SPLINE
SPL {X  -106.708, Y  +258.294, Z    +0.000, E1   +53.789, E3 +25392.422}
SPL {X  -137.973, Y  +296.505, Z    +0.000, E1   +48.844, E3 +25431.202}
SPL {X  -154.359, Y  +335.426, Z    +0.000, E1   +34.338, E3 +25444.098}
SPL {X  -159.279, Y  +362.429, Z    +0.000, E1   +16.013, E3 +25447.698}
SPL {X  -159.976, Y  +375.387, Z    +0.000, E1    +4.229, E3 +25448.348}
SPL {X  -159.990, Y  +379.485, Z    +0.000, E1    +0.028, E3 +25448.394}
SPL {X  -159.990, Y  +381.270, Z    +0.000, E1    -3.383, E3 +25448.411}
SPL {X  -159.990, Y  +384.811, Z    +0.000, E1   -11.531, E3 +25448.501}
SPL {X  -159.990, Y  +388.002, Z    +0.000, E1   -19.281, E3 +25448.651}
SPL {X  -159.990, Y  +394.075, Z    +0.000, E1   -32.836, E3 +25449.129}
SPL {X  -159.990, Y  +405.152, Z    +0.000, E1   -50.697, E3 +25450.553}
SPL {X  -159.990, Y  +423.293, Z    +0.000, E1   -63.280, E3 +25454.554}
SPL {X  -159.990, Y  +493.649, Z    +0.000, E1   -71.671, E3 +25480.258}
SPL {X  -159.990, Y  +662.531, Z    +0.000, E1   -73.010, E3 +25567.081}
SPL {X  -159.805, Y  +684.185, Z    +0.000, E1   -72.979, E3 +25581.365}
SPL {X  -158.739, Y  +696.464, Z    +0.000, E1   -72.862, E3 +25590.484}
SPL {X  -156.417, Y  +710.124, Z    +0.000, E1   -72.650, E3 +25601.707}
SPL {X  -153.206, Y  +722.596, Z    +0.000, E1   -72.287, E3 +25613.146}
SPL {X  -150.445, Y  +730.933, Z    +0.000, E1   -71.979, E3 +25621.356}
SPL {X  -147.389, Y  +738.737, Z    +0.000, E1   -71.634, E3 +25629.429}
SPL {X  -144.044, Y  +746.129, Z    +0.000, E1   -71.236, E3 +25637.423}
SPL {X  -140.684, Y  +752.689, Z    +0.000, E1   -70.820, E3 +25644.798}
SPL {X  -137.335, Y  +758.572, Z    +0.000, E1   -70.388, E3 +25651.606}
SPL {X  -134.566, Y  +763.037, Z    +0.000, E1   -70.007, E3 +25656.902}
SPL {X  -131.456, Y  +767.693, Z    +0.000, E1   -69.587, E3 +25662.465}
SPL {X  -127.440, Y  +773.226, Z    +0.000, E1   -69.006, E3 +25669.149}
SPL {X  -123.127, Y  +778.659, Z    +0.000, E1   -68.349, E3 +25675.691}
SPL {X   -80.879, Y  +814.541, Z    +0.000, E1   -55.704, E3 +25798.595}
ENDSPLINE

SPLINE
SPL {X  -125.518, Y  +775.707, Z    +0.000, E1   -52.189, E3 +25970.073}
SPL {X  -150.797, Y  +729.951, Z    +0.000, E1   -39.777, E3 +25992.808}
SPL {X  -158.456, Y  +698.602, Z    +0.000, E1   -21.523, E3 +25998.510}
SPL {X  -159.738, Y  +685.469, Z    +0.000, E1   -10.595, E3 +25999.565}
SPL {X  -159.986, Y  +677.650, Z    +0.000, E1    -3.291, E3 +25999.819}
SPL {X  -159.990, Y  +674.500, Z    +0.000, E1    +0.000, E3 +25999.850}
SPL {X  -159.990, Y  +672.716, Z    +0.000, E1    +3.405, E3 +25999.866}
SPL {X  -159.990, Y  +668.521, Z    +0.000, E1   +13.007, E3 +25999.985}
SPL {X  -159.990, Y  +662.839, Z    +0.000, E1   +26.519, E3 +26000.328}
SPL {X  -159.990, Y  +653.836, Z    +0.000, E1   +43.967, E3 +26001.258}
SPL {X  -159.990, Y  +641.022, Z    +0.000, E1   +57.726, E3 +26003.567}
SPL {X  -159.990, Y  +617.987, Z    +0.000, E1   +67.134, E3 +26009.463}
SPL {X  -159.990, Y  +532.407, Z    +0.000, E1   +73.084, E3 +26040.369}
SPL {X  -159.990, Y  +382.957, Z    +0.000, E1   +73.647, E3 +26116.629}
SPL {X  -159.615, Y  +366.548, Z    +0.000, E1   +73.602, E3 +26127.271}
SPL {X  -157.928, Y  +351.899, Z    +0.000, E1   +73.451, E3 +26138.126}
ENDSPLINE

SPLINE
SPL {X  -159.990, Y  +380.170, Z    +0.000, E1   +69.785, E3 +26154.266}
ENDSPLINE

SPLINE
SPL {X  -158.227, Y  +353.814, Z    +0.000, E1   +70.663, E3 +26166.159}
SPL {X  -155.560, Y  +340.111, Z    +0.000, E1   +70.976, E3 +26173.181}
SPL {X  -151.918, Y  +327.322, Z    +0.000, E1   +71.266, E3 +26179.525}
SPL {X  -144.697, Y  +309.238, Z    +0.000, E1   +71.848, E3 +26186.475}
SPL {X  -140.298, Y  +300.601, Z    +0.000, E1   +71.461, E3 +26194.762}
SPL {X  -137.001, Y  +294.872, Z    +0.000, E1   +71.048, E3 +26201.270}
SPL {X  -133.301, Y  +289.026, Z    +0.000, E1   +70.567, E3 +26208.057}
SPL {X  -128.648, Y  +282.387, Z    +0.000, E1   +69.939, E3 +26215.872}
SPL {X  -125.063, Y  +277.720, Z    +0.000, E1   +69.378, E3 +26221.448}
SPL {X  -122.086, Y  +274.099, Z    +0.000, E1   +68.932, E3 +26225.693}
SPL {X   -84.117, Y  +241.407, Z    +0.000, E1   +58.224, E3 +26316.576}
ENDSPLINE

SPLINE
SPL {X  -106.708, Y  +258.294, Z    +0.000, E1   +53.789, E3 +26495.363}
SPL {X  -137.973, Y  +296.505, Z    +0.000, E1   +48.844, E3 +26534.143}
SPL {X  -154.359, Y  +335.426, Z    +0.000, E1   +34.338, E3 +26547.039}
SPL {X  -159.279, Y  +362.429, Z    +0.000, E1   +16.013, E3 +26550.639}
SPL {X  -159.976, Y  +375.387, Z    +0.000, E1    +4.229, E3 +26551.290}
SPL {X  -159.990, Y  +379.485, Z    +0.000, E1    +0.028, E3 +26551.335}
SPL {X  -159.990, Y  +381.270, Z    +0.000, E1    -3.383, E3 +26551.352}
SPL {X  -159.990, Y  +384.811, Z    +0.000, E1   -11.531, E3 +26551.442}
SPL {X  -159.990, Y  +390.180, Z    +0.000, E1   -24.142, E3 +26551.745}
SPL {X  -159.990, Y  +397.074, Z    +0.000, E1   -39.012, E3 +26552.355}
SPL {X  -159.990, Y  +405.152, Z    +0.000, E1   -50.697, E3 +26553.494}
SPL {X  -159.990, Y  +423.293, Z    +0.000, E1   -63.280, E3 +26557.496}
SPL {X  -159.990, Y  +493.649, Z    +0.000, E1   -71.671, E3 +26583.199}
SPL {X  -159.990, Y  +654.929, Z    +0.000, E1   -72.988, E3 +26665.149}
SPL {X  -159.990, Y  +668.018, Z    +0.000, E1   -72.989, E3 +26673.642}
SPL {X  -159.805, Y  +684.185, Z    +0.000, E1   -72.979, E3 +26684.307}
SPL {X  -158.295, Y  +699.729, Z    +0.000, E1   -72.830, E3 +26695.977}
SPL {X  -155.857, Y  +712.630, Z    +0.000, E1   -72.572, E3 +26706.906}
SPL {X  -153.206, Y  +722.596, Z    +0.000, E1   -72.287, E3 +26716.087}
SPL {X  -150.445, Y  +730.933, Z    +0.000, E1   -71.979, E3 +26724.297}
SPL {X  -147.389, Y  +738.737, Z    +0.000, E1   -71.634, E3 +26732.370}
SPL {X  -144.044, Y  +746.129, Z    +0.000, E1   -71.236, E3 +26740.364}
SPL {X  -140.684, Y  +752.689, Z    +0.000, E1   -70.820, E3 +26747.740}
SPL {X  -137.335, Y  +758.572, Z    +0.000, E1   -70.388, E3 +26754.547}
SPL {X  -133.651, Y  +764.444, Z    +0.000, E1   -69.897, E3 +26761.499}
SPL {X  -130.650, Y  +768.844, Z    +0.000, E1   -69.455, E3 +26766.820}
SPL {X  -127.440, Y  +773.226, Z    +0.000, E1   -69.006, E3 +26772.090}
SPL {X  -123.127, Y  +778.659, Z    +0.000, E1   -68.349, E3 +26778.632}
SPL {X   -80.879, Y  +814.541, Z    +0.000, E1   -55.704, E3 +26901.536}
ENDSPLINE

SPLINE
SPL {X  -125.518, Y  +775.707, Z    +0.000, E1   -52.189, E3 +27073.014}
SPL {X  -150.797, Y  +729.951, Z    +0.000, E1   -39.777, E3 +27095.749}
SPL {X  -157.402, Y  +705.160, Z    +0.000, E1   -26.108, E3 +27100.701}
SPL {X  -159.480, Y  +689.270, Z    +0.000, E1   -14.023, E3 +27102.266}
SPL {X  -159.986, Y  +677.650, Z    +0.000, E1    -3.291, E3 +27102.761}
SPL {X  -159.990, Y  +674.500, Z    +0.000, E1    +0.000, E3 +27102.791}
SPL {X  -159.990, Y  +672.716, Z    +0.000, E1    +3.405, E3 +27102.808}
SPL {X  -159.990, Y  +668.521, Z    +0.000, E1   +13.007, E3 +27102.927}
SPL {X  -159.990, Y  +664.286, Z    +0.000, E1   +23.338, E3 +27103.158}
SPL {X  -159.990, Y  +658.431, Z    +0.000, E1   +35.998, E3 +27103.653}
SPL {X  -159.990, Y  +650.524, Z    +0.000, E1   +48.779, E3 +27104.641}
SPL {X  -159.990, Y  +641.022, Z    +0.000, E1   +57.726, E3 +27106.508}
SPL {X  -159.990, Y  +617.987, Z    +0.000, E1   +67.134, E3 +27112.404}
SPL {X  -159.990, Y  +532.407, Z    +0.000, E1   +73.084, E3 +27143.310}
SPL {X  -159.990, Y  +390.607, Z    +0.000, E1   +73.632, E3 +27214.847}
SPL {X  -159.886, Y  +371.742, Z    +0.000, E1   +73.650, E3 +27226.633}
SPL {X  -157.928, Y  +351.899, Z    +0.000, E1   +73.451, E3 +27241.067}
ENDSPLINE

SPLINE
SPL {X  -159.990, Y  +380.170, Z    +0.000, E1   +69.785, E3 +27257.207}
ENDSPLINE

SPLINE
SPL {X  -158.227, Y  +353.814, Z    +0.000, E1   +70.663, E3 +27269.101}
SPL {X  -154.257, Y  +335.055, Z    +0.000, E1   +71.089, E3 +27278.729}
SPL {X  -148.153, Y  +317.104, Z    +0.000, E1   +71.658, E3 +27285.874}
SPL {X  -143.479, Y  +306.716, Z    +0.000, E1   +71.847, E3 +27290.948}
SPL {X  -140.298, Y  +300.601, Z    +0.000, E1   +71.461, E3 +27297.703}
SPL {X  -137.001, Y  +294.872, Z    +0.000, E1   +71.048, E3 +27304.212}
SPL {X  -133.301, Y  +289.026, Z    +0.000, E1   +70.567, E3 +27310.998}
SPL {X  -129.603, Y  +283.692, Z    +0.000, E1   +70.051, E3 +27317.298}
SPL {X  -125.807, Y  +278.659, Z    +0.000, E1   +69.508, E3 +27323.257}
SPL {X  -122.086, Y  +274.099, Z    +0.000, E1   +68.932, E3 +27328.634}
SPL {X   -84.117, Y  +241.407, Z    +0.000, E1   +58.224, E3 +27419.517}
ENDSPLINE

SPLINE
SPL {X  -116.986, Y  +268.362, Z    +0.000, E1   +53.233, E3 +27613.432}
SPL {X  -146.319, Y  +312.789, Z    +0.000, E1   +44.152, E3 +27643.899}
SPL {X  -157.053, Y  +346.986, Z    +0.000, E1   +27.437, E3 +27651.930}
SPL {X  -159.518, Y  +365.226, Z    +0.000, E1   +13.562, E3 +27653.795}
SPL {X  -159.976, Y  +375.387, Z    +0.000, E1    +4.229, E3 +27654.231}
SPL {X  -159.990, Y  +379.485, Z    +0.000, E1    +0.028, E3 +27654.276}
SPL {X  -159.990, Y  +381.270, Z    +0.000, E1    -3.383, E3 +27654.293}
SPL {X  -159.990, Y  +384.811, Z    +0.000, E1   -11.531, E3 +27654.383}
SPL {X  -159.990, Y  +390.180, Z    +0.000, E1   -24.142, E3 +27654.686}
SPL {X  -159.990, Y  +397.074, Z    +0.000, E1   -39.012, E3 +27655.296}
SPL {X  -159.990, Y  +405.152, Z    +0.000, E1   -50.697, E3 +27656.435}
SPL {X  -159.990, Y  +423.293, Z    +0.000, E1   -63.280, E3 +27660.437}
SPL {X  -159.990, Y  +493.649, Z    +0.000, E1   -71.671, E3 +27686.141}
SPL {X  -159.990, Y  +662.531, Z    +0.000, E1   -73.010, E3 +27772.964}
SPL {X  -159.805, Y  +684.185, Z    +0.000, E1   -72.979, E3 +27787.248}
SPL {X  -158.295, Y  +699.729, Z    +0.000, E1   -72.830, E3 +27798.918}
SPL {X  -155.857, Y  +712.630, Z    +0.000, E1   -72.572, E3 +27809.847}
SPL {X  -153.206, Y  +722.596, Z    +0.000, E1   -72.287, E3 +27819.028}
SPL {X  -150.445, Y  +730.933, Z    +0.000, E1   -71.979, E3 +27827.238}
SPL {X  -147.389, Y  +738.737, Z    +0.000, E1   -71.634, E3 +27835.311}
SPL {X  -144.044, Y  +746.129, Z    +0.000, E1   -71.236, E3 +27843.305}
SPL {X  -140.684, Y  +752.689, Z    +0.000, E1   -70.820, E3 +27850.681}
SPL {X  -137.335, Y  +758.572, Z    +0.000, E1   -70.388, E3 +27857.488}
SPL {X  -133.651, Y  +764.444, Z    +0.000, E1   -69.897, E3 +27864.440}
SPL {X  -129.492, Y  +770.461, Z    +0.000, E1   -69.311, E3 +27871.680}
SPL {X  -125.168, Y  +776.148, Z    +0.000, E1   -68.666, E3 +27878.557}
SPL {X  -122.036, Y  +779.960, Z    +0.000, E1   -68.144, E3 +27883.160}
SPL {X   -80.879, Y  +814.541, Z    +0.000, E1   -55.704, E3 +28004.478}
ENDSPLINE

SPLINE
SPL {X  -125.518, Y  +775.707, Z    +0.000, E1   -52.189, E3 +28175.955}
SPL {X  -144.748, Y  +744.653, Z    +0.000, E1   -45.208, E3 +28194.151}
SPL {X  -153.147, Y  +722.791, Z    +0.000, E1   -36.417, E3 +28200.547}
SPL {X  -157.402, Y  +705.160, Z    +0.000, E1   -26.108, E3 +28203.642}
SPL {X  -159.480, Y  +689.270, Z    +0.000, E1   -14.023, E3 +28205.208}
SPL {X  -159.986, Y  +677.650, Z    +0.000, E1    -3.291, E3 +28205.702}
SPL {X  -159.990, Y  +674.500, Z    +0.000, E1    +0.000, E3 +28205.732}
SPL {X  -159.990, Y  +672.716, Z    +0.000, E1    +3.405, E3 +28205.749}
SPL {X  -159.990, Y  +668.521, Z    +0.000, E1   +13.007, E3 +28205.868}
SPL {X  -159.990, Y  +664.286, Z    +0.000, E1   +23.338, E3 +28206.099}
SPL {X  -159.990, Y  +658.431, Z    +0.000, E1   +35.998, E3 +28206.594}
SPL {X  -159.990, Y  +650.524, Z    +0.000, E1   +48.779, E3 +28207.582}
SPL {X  -159.990, Y  +641.022, Z    +0.000, E1   +57.726, E3 +28209.449}
SPL {X  -159.990, Y  +617.987, Z    +0.000, E1   +67.134, E3 +28215.345}
SPL {X  -159.990, Y  +532.407, Z    +0.000, E1   +73.084, E3 +28246.252}
SPL {X  -159.990, Y  +390.607, Z    +0.000, E1   +73.632, E3 +28317.788}
SPL {X  -159.886, Y  +371.742, Z    +0.000, E1   +73.650, E3 +28329.574}
SPL {X  -157.928, Y  +351.899, Z    +0.000, E1   +73.451, E3 +28344.008}
ENDSPLINE

SPLINE
SPL {X  -159.990, Y  +380.170, Z    +0.000, E1   +69.785, E3 +28360.148}
ENDSPLINE

SPLINE
SPL {X  -158.227, Y  +353.814, Z    +0.000, E1   +70.663, E3 +28372.042}
SPL {X  -155.560, Y  +340.111, Z    +0.000, E1   +70.976, E3 +28379.064}
SPL {X  -151.918, Y  +327.322, Z    +0.000, E1   +71.266, E3 +28385.407}
SPL {X  -144.697, Y  +309.238, Z    +0.000, E1   +71.848, E3 +28392.357}
SPL {X  -140.298, Y  +300.601, Z    +0.000, E1   +71.461, E3 +28400.644}
SPL {X  -137.001, Y  +294.872, Z    +0.000, E1   +71.048, E3 +28407.153}
SPL {X  -133.301, Y  +289.026, Z    +0.000, E1   +70.567, E3 +28413.939}
SPL {X  -129.603, Y  +283.692, Z    +0.000, E1   +70.051, E3 +28420.239}
SPL {X  -125.807, Y  +278.659, Z    +0.000, E1   +69.508, E3 +28426.198}
SPL {X  -122.086, Y  +274.099, Z    +0.000, E1   +68.932, E3 +28431.576}
SPL {X   -84.117, Y  +241.407, Z    +0.000, E1   +58.224, E3 +28522.458}
ENDSPLINE

SPLINE
SPL {X  -106.708, Y  +258.294, Z    +0.000, E1   +53.789, E3 +28701.245}
SPL {X  -137.973, Y  +296.505, Z    +0.000, E1   +48.844, E3 +28740.025}
SPL {X  -154.359, Y  +335.426, Z    +0.000, E1   +34.338, E3 +28752.921}
SPL {X  -159.279, Y  +362.429, Z    +0.000, E1   +16.013, E3 +28756.521}
SPL {X  -159.976, Y  +375.387, Z    +0.000, E1    +4.229, E3 +28757.172}
SPL {X  -159.990, Y  +379.485, Z    +0.000, E1    +0.028, E3 +28757.217}
SPL {X  -159.990, Y  +381.270, Z    +0.000, E1    -3.383, E3 +28757.234}
SPL {X  -159.990, Y  +386.246, Z    +0.000, E1   -14.704, E3 +28757.392}
SPL {X  -159.990, Y  +394.075, Z    +0.000, E1   -32.836, E3 +28757.952}
SPL {X  -159.990, Y  +405.152, Z    +0.000, E1   -50.697, E3 +28759.377}
SPL {X  -159.990, Y  +423.293, Z    +0.000, E1   -63.280, E3 +28763.378}
SPL {X  -159.990, Y  +493.649, Z    +0.000, E1   -71.671, E3 +28789.082}
SPL {X  -159.990, Y  +662.531, Z    +0.000, E1   -73.010, E3 +28875.905}
SPL {X  -159.805, Y  +684.185, Z    +0.000, E1   -72.979, E3 +28890.189}
SPL {X  -158.295, Y  +699.729, Z    +0.000, E1   -72.830, E3 +28901.859}
SPL {X  -155.857, Y  +712.630, Z    +0.000, E1   -72.572, E3 +28912.788}
SPL {X  -153.206, Y  +722.596, Z    +0.000, E1   -72.287, E3 +28921.969}
SPL {X  -150.445, Y  +730.933, Z    +0.000, E1   -71.979, E3 +28930.179}
SPL {X  -147.389, Y  +738.737, Z    +0.000, E1   -71.634, E3 +28938.252}
SPL {X  -144.044, Y  +746.129, Z    +0.000, E1   -71.236, E3 +28946.247}
SPL {X  -140.684, Y  +752.689, Z    +0.000, E1   -70.820, E3 +28953.622}
SPL {X  -136.099, Y  +760.606, Z    +0.000, E1   -70.253, E3 +28962.777}
SPL {X  -131.456, Y  +767.693, Z    +0.000, E1   -69.587, E3 +28971.289}
SPL {X  -127.440, Y  +773.226, Z    +0.000, E1   -69.006, E3 +28977.973}
SPL {X  -123.127, Y  +778.659, Z    +0.000, E1   -68.349, E3 +28984.515}
SPL {X   -80.879, Y  +814.541, Z    +0.000, E1   -55.704, E3 +29107.419}
ENDSPLINE

SPLINE
SPL {X  -125.518, Y  +775.707, Z    +0.000, E1   -52.189, E3 +29278.896}
SPL {X  -150.797, Y  +729.951, Z    +0.000, E1   -39.777, E3 +29301.631}
SPL {X  -157.402, Y  +705.160, Z    +0.000, E1   -26.108, E3 +29306.583}
SPL {X  -159.480, Y  +689.270, Z    +0.000, E1   -14.023, E3 +29308.149}
SPL {X  -159.986, Y  +677.650, Z    +0.000, E1    -3.291, E3 +29308.643}
SPL {X  -159.990, Y  +674.500, Z    +0.000, E1    +0.000, E3 +29308.673}
SPL {X  -159.990, Y  +672.716, Z    +0.000, E1    +3.405, E3 +29308.690}
SPL {X  -159.990, Y  +668.521, Z    +0.000, E1   +13.007, E3 +29308.809}
SPL {X  -159.990, Y  +662.839, Z    +0.000, E1   +26.519, E3 +29309.151}
SPL {X  -159.990, Y  +653.836, Z    +0.000, E1   +43.967, E3 +29310.082}
SPL {X  -159.990, Y  +641.022, Z    +0.000, E1   +57.726, E3 +29312.391}
SPL {X  -159.990, Y  +617.987, Z    +0.000, E1   +67.134, E3 +29318.286}
SPL {X  -159.990, Y  +532.407, Z    +0.000, E1   +73.084, E3 +29349.193}
SPL {X  -159.990, Y  +390.607, Z    +0.000, E1   +73.632, E3 +29420.729}
SPL {X  -159.886, Y  +371.742, Z    +0.000, E1   +73.650, E3 +29432.516}
SPL {X  -157.928, Y  +351.899, Z    +0.000, E1   +73.451, E3 +29446.949}
ENDSPLINE

SPLINE
SPL {X  -159.990, Y  +380.170, Z    +0.000, E1   +69.785, E3 +29463.089}
ENDSPLINE

SPLINE
SPL {X  -158.227, Y  +353.814, Z    +0.000, E1   +70.663, E3 +29474.983}
SPL {X  -155.560, Y  +340.111, Z    +0.000, E1   +70.976, E3 +29482.005}
SPL {X  -151.918, Y  +327.322, Z    +0.000, E1   +71.266, E3 +29488.349}
SPL {X  -144.697, Y  +309.238, Z    +0.000, E1   +71.848, E3 +29495.298}
SPL {X  -140.298, Y  +300.601, Z    +0.000, E1   +71.461, E3 +29503.586}
SPL {X  -135.903, Y  +293.078, Z    +0.000, E1   +70.930, E3 +29512.123}
SPL {X  -130.487, Y  +284.926, Z    +0.000, E1   +70.202, E3 +29521.683}
SPL {X  -125.807, Y  +278.659, Z    +0.000, E1   +69.508, E3 +29529.139}
SPL {X  -122.967, Y  +275.148, Z    +0.000, E1   +69.053, E3 +29533.308}
SPL {X  -121.236, Y  +273.103, Z    +0.000, E1   +68.779, E3 +29535.694}
SPL {X   -84.117, Y  +241.407, Z    +0.000, E1   +58.224, E3 +29625.399}
ENDSPLINE

SPLINE
SPL {X  -116.986, Y  +268.362, Z    +0.000, E1   +53.233, E3 +29819.315}
SPL {X  -146.319, Y  +312.789, Z    +0.000, E1   +44.152, E3 +29849.781}
SPL {X  -157.053, Y  +346.986, Z    +0.000, E1   +27.437, E3 +29857.812}
SPL {X  -159.518, Y  +365.226, Z    +0.000, E1   +13.562, E3 +29859.678}
SPL {X  -159.976, Y  +375.387, Z    +0.000, E1    +4.229, E3 +29860.113}
SPL {X  -159.990, Y  +379.485, Z    +0.000, E1    +0.028, E3 +29860.158}
SPL {X  -159.990, Y  +381.270, Z    +0.000, E1    -3.383, E3 +29860.175}
SPL {X  -159.990, Y  +386.246, Z    +0.000, E1   -14.704, E3 +29860.333}
SPL {X  -159.990, Y  +394.075, Z    +0.000, E1   -32.836, E3 +29860.894}
SPL {X  -159.990, Y  +405.152, Z    +0.000, E1   -50.697, E3 +29862.318}
SPL {X  -159.990, Y  +423.293, Z    +0.000, E1   -63.280, E3 +29866.319}
SPL {X  -159.990, Y  +493.649, Z    +0.000, E1   -71.671, E3 +29892.023}
SPL {X  -159.990, Y  +662.531, Z    +0.000, E1   -73.010, E3 +29978.846}
SPL {X  -159.805, Y  +684.185, Z    +0.000, E1   -72.979, E3 +29993.130}
SPL {X  -158.295, Y  +699.729, Z    +0.000, E1   -72.830, E3 +30004.800}
SPL {X  -155.857, Y  +712.630, Z    +0.000, E1   -72.572, E3 +30015.729}
SPL {X  -153.206, Y  +722.596, Z    +0.000, E1   -72.287, E3 +30024.910}
SPL {X  -150.445, Y  +730.933, Z    +0.000, E1   -71.979, E3 +30033.121}
SPL {X  -147.389, Y  +738.737, Z    +0.000, E1   -71.634, E3 +30041.193}
SPL {X  -144.044, Y  +746.129, Z    +0.000, E1   -71.236, E3 +30049.188}
SPL {X  -140.684, Y  +752.689, Z    +0.000, E1   -70.820, E3 +30056.563}
SPL {X  -136.099, Y  +760.606, Z    +0.000, E1   -70.253, E3 +30065.718}
SPL {X  -131.456, Y  +767.693, Z    +0.000, E1   -69.587, E3 +30074.230}
SPL {X  -127.440, Y  +773.226, Z    +0.000, E1   -69.006, E3 +30080.914}
SPL {X  -123.127, Y  +778.659, Z    +0.000, E1   -68.349, E3 +30087.456}
SPL {X   -80.879, Y  +814.541, Z    +0.000, E1   -55.704, E3 +30210.360}
ENDSPLINE

SPLINE
SPL {X  -125.518, Y  +775.707, Z    +0.000, E1   -52.189, E3 +30381.837}
SPL {X  -150.797, Y  +729.951, Z    +0.000, E1   -39.777, E3 +30404.572}
SPL {X  -158.456, Y  +698.602, Z    +0.000, E1   -21.523, E3 +30410.275}
SPL {X  -159.738, Y  +685.469, Z    +0.000, E1   -10.595, E3 +30411.329}
SPL {X  -159.986, Y  +677.650, Z    +0.000, E1    -3.291, E3 +30411.584}
SPL {X  -159.990, Y  +674.500, Z    +0.000, E1    +0.000, E3 +30411.615}
SPL {X  -159.990, Y  +672.716, Z    +0.000, E1    +3.405, E3 +30411.631}
SPL {X  -159.990, Y  +668.521, Z    +0.000, E1   +13.007, E3 +30411.750}
SPL {X  -159.990, Y  +662.839, Z    +0.000, E1   +26.519, E3 +30412.093}
SPL {X  -159.990, Y  +653.836, Z    +0.000, E1   +43.967, E3 +30413.023}
SPL {X  -159.990, Y  +641.022, Z    +0.000, E1   +57.726, E3 +30415.332}
SPL {X  -159.990, Y  +617.987, Z    +0.000, E1   +67.134, E3 +30421.227}
SPL {X  -159.990, Y  +532.407, Z    +0.000, E1   +73.084, E3 +30452.134}
SPL {X  -159.990, Y  +382.957, Z    +0.000, E1   +73.647, E3 +30528.394}
SPL {X  -159.615, Y  +366.548, Z    +0.000, E1   +73.602, E3 +30539.036}
SPL {X  -157.928, Y  +351.899, Z    +0.000, E1   +73.451, E3 +30549.890}
ENDSPLINE

SPLINE
SPL {X  -159.990, Y  +380.170, Z    +0.000, E1   +69.785, E3 +30566.031}
ENDSPLINE

SPLINE
SPL {X  -158.227, Y  +353.814, Z    +0.000, E1   +70.663, E3 +30577.924}
SPL {X  -154.257, Y  +335.055, Z    +0.000, E1   +71.089, E3 +30587.552}
SPL {X  -148.153, Y  +317.104, Z    +0.000, E1   +71.658, E3 +30594.698}
SPL {X  -143.479, Y  +306.716, Z    +0.000, E1   +71.847, E3 +30599.771}
SPL {X  -140.298, Y  +300.601, Z    +0.000, E1   +71.461, E3 +30606.527}
SPL {X  -137.001, Y  +294.872, Z    +0.000, E1   +71.048, E3 +30613.035}
SPL {X  -133.301, Y  +289.026, Z    +0.000, E1   +70.567, E3 +30619.822}
SPL {X  -128.648, Y  +282.387, Z    +0.000, E1   +69.939, E3 +30627.637}
SPL {X  -125.063, Y  +277.720, Z    +0.000, E1   +69.378, E3 +30633.213}
SPL {X  -122.086, Y  +274.099, Z    +0.000, E1   +68.932, E3 +30637.458}
SPL {X   -84.117, Y  +241.407, Z    +0.000, E1   +58.224, E3 +30728.341}
ENDSPLINE

SPLINE
SPL {X  -106.708, Y  +258.294, Z    +0.000, E1   +53.789, E3 +30907.127}
SPL {X  -137.973, Y  +296.505, Z    +0.000, E1   +48.844, E3 +30945.908}
SPL {X  -154.359, Y  +335.426, Z    +0.000, E1   +34.338, E3 +30958.804}
SPL {X  -159.279, Y  +362.429, Z    +0.000, E1   +16.013, E3 +30962.404}
SPL {X  -159.976, Y  +375.387, Z    +0.000, E1    +4.229, E3 +30963.054}
SPL {X  -159.990, Y  +379.485, Z    +0.000, E1    +0.028, E3 +30963.099}
SPL {X  -159.990, Y  +381.270, Z    +0.000, E1    -3.383, E3 +30963.117}
SPL {X  -159.990, Y  +384.811, Z    +0.000, E1   -11.531, E3 +30963.207}
SPL {X  -159.990, Y  +390.180, Z    +0.000, E1   -24.142, E3 +30963.510}
SPL {X  -159.990, Y  +397.074, Z    +0.000, E1   -39.012, E3 +30964.120}
SPL {X  -159.990, Y  +405.152, Z    +0.000, E1   -50.697, E3 +30965.259}
SPL {X  -159.990, Y  +423.293, Z    +0.000, E1   -63.280, E3 +30969.260}
SPL {X  -159.990, Y  +493.649, Z    +0.000, E1   -71.671, E3 +30994.964}
SPL {X  -159.990, Y  +662.531, Z    +0.000, E1   -73.010, E3 +31081.787}
SPL {X  -159.805, Y  +684.185, Z    +0.000, E1   -72.979, E3 +31096.071}
SPL {X  -158.739, Y  +696.464, Z    +0.000, E1   -72.862, E3 +31105.190}
SPL {X  -156.417, Y  +710.124, Z    +0.000, E1   -72.650, E3 +31116.413}
SPL {X  -153.206, Y  +722.596, Z    +0.000, E1   -72.287, E3 +31127.851}
SPL {X  -150.445, Y  +730.933, Z    +0.000, E1   -71.979, E3 +31136.062}
SPL {X  -147.389, Y  +738.737, Z    +0.000, E1   -71.634, E3 +31144.135}
SPL {X  -144.044, Y  +746.129, Z    +0.000, E1   -71.236, E3 +31152.129}
SPL {X  -140.684, Y  +752.689, Z    +0.000, E1   -70.820, E3 +31159.504}
SPL {X  -137.335, Y  +758.572, Z    +0.000, E1   -70.388, E3 +31166.311}
SPL {X  -134.566, Y  +763.037, Z    +0.000, E1   -70.007, E3 +31171.608}
SPL {X  -131.456, Y  +767.693, Z    +0.000, E1   -69.587, E3 +31177.171}
SPL {X  -127.440, Y  +773.226, Z    +0.000, E1   -69.006, E3 +31183.855}
SPL {X  -123.127, Y  +778.659, Z    +0.000, E1   -68.349, E3 +31190.397}
SPL {X   -80.879, Y  +814.541, Z    +0.000, E1   -55.704, E3 +31313.301}
ENDSPLINE

SPLINE
SPL {X  -125.518, Y  +775.707, Z    +0.000, E1   -52.189, E3 +31484.779}
SPL {X  -144.748, Y  +744.653, Z    +0.000, E1   -45.208, E3 +31502.974}
SPL {X  -153.147, Y  +722.791, Z    +0.000, E1   -36.417, E3 +31509.370}
SPL {X  -157.402, Y  +705.160, Z    +0.000, E1   -26.108, E3 +31512.465}
SPL {X  -159.480, Y  +689.270, Z    +0.000, E1   -14.023, E3 +31514.031}
SPL {X  -159.986, Y  +677.650, Z    +0.000, E1    -3.291, E3 +31514.525}
SPL {X  -159.990, Y  +674.500, Z    +0.000, E1    +0.000, E3 +31514.556}
SPL {X  -159.990, Y  +672.716, Z    +0.000, E1    +3.405, E3 +31514.572}
SPL {X  -159.990, Y  +668.521, Z    +0.000, E1   +13.007, E3 +31514.691}
SPL {X  -159.990, Y  +662.839, Z    +0.000, E1   +26.519, E3 +31515.034}
SPL {X  -159.990, Y  +653.836, Z    +0.000, E1   +43.967, E3 +31515.964}
SPL {X  -159.990, Y  +641.022, Z    +0.000, E1   +57.726, E3 +31518.273}
SPL {X  -159.990, Y  +617.987, Z    +0.000, E1   +67.134, E3 +31524.168}
SPL {X  -159.990, Y  +532.407, Z    +0.000, E1   +73.084, E3 +31555.075}
SPL {X  -159.990, Y  +382.957, Z    +0.000, E1   +73.647, E3 +31631.335}
SPL {X  -159.615, Y  +366.548, Z    +0.000, E1   +73.602, E3 +31641.977}
SPL {X  -157.928, Y  +351.899, Z    +0.000, E1   +73.451, E3 +31652.832}
ENDSPLINE

SPLINE
SPL {X  -159.990, Y  +380.170, Z    +0.000, E1   +69.785, E3 +31668.972}
ENDSPLINE

SPLINE
SPL {X  -158.227, Y  +353.814, Z    +0.000, E1   +70.663, E3 +31680.865}
SPL {X  -155.560, Y  +340.111, Z    +0.000, E1   +70.976, E3 +31687.887}
SPL {X  -151.918, Y  +327.322, Z    +0.000, E1   +71.266, E3 +31694.231}
SPL {X  -144.697, Y  +309.238, Z    +0.000, E1   +71.848, E3 +31701.181}
SPL {X  -140.298, Y  +300.601, Z    +0.000, E1   +71.461, E3 +31709.468}
SPL {X  -135.903, Y  +293.078, Z    +0.000, E1   +70.930, E3 +31718.006}
SPL {X  -130.487, Y  +284.926, Z    +0.000, E1   +70.202, E3 +31727.565}
SPL {X  -125.807, Y  +278.659, Z    +0.000, E1   +69.508, E3 +31735.022}
SPL {X  -122.967, Y  +275.148, Z    +0.000, E1   +69.053, E3 +31739.190}
SPL {X  -121.236, Y  +273.103, Z    +0.000, E1   +68.779, E3 +31741.576}
SPL {X   -84.117, Y  +241.407, Z    +0.000, E1   +58.224, E3 +31831.282}
ENDSPLINE

SPLINE
SPL {X  -106.708, Y  +258.294, Z    +0.000, E1   +53.789, E3 +32010.069}
SPL {X  -137.973, Y  +296.505, Z    +0.000, E1   +48.844, E3 +32048.849}
SPL {X  -150.692, Y  +323.752, Z    +0.000, E1   +39.895, E3 +32059.214}
SPL {X  -157.053, Y  +346.986, Z    +0.000, E1   +27.437, E3 +32063.695}
SPL {X  -159.518, Y  +365.226, Z    +0.000, E1   +13.562, E3 +32065.560}
SPL {X  -159.976, Y  +375.387, Z    +0.000, E1    +4.229, E3 +32065.996}
SPL {X  -159.990, Y  +379.485, Z    +0.000, E1    +0.028, E3 +32066.041}
SPL {X  -159.990, Y  +381.270, Z    +0.000, E1    -3.383, E3 +32066.058}
SPL {X  -159.990, Y  +384.811, Z    +0.000, E1   -11.531, E3 +32066.148}
SPL {X  -159.990, Y  +390.180, Z    +0.000, E1   -24.142, E3 +32066.451}
SPL {X  -159.990, Y  +397.074, Z    +0.000, E1   -39.012, E3 +32067.061}
SPL {X  -159.990, Y  +405.152, Z    +0.000, E1   -50.697, E3 +32068.200}
SPL {X  -159.990, Y  +423.293, Z    +0.000, E1   -63.280, E3 +32072.201}
SPL {X  -159.990, Y  +493.649, Z    +0.000, E1   -71.671, E3 +32097.905}
SPL {X  -159.990, Y  +662.531, Z    +0.000, E1   -73.010, E3 +32184.728}
SPL {X  -159.805, Y  +684.185, Z    +0.000, E1   -72.979, E3 +32199.012}
SPL {X  -158.739, Y  +696.464, Z    +0.000, E1   -72.862, E3 +32208.131}
SPL {X  -156.417, Y  +710.124, Z    +0.000, E1   -72.650, E3 +32219.355}
SPL {X  -153.206, Y  +722.596, Z    +0.000, E1   -72.287, E3 +32230.793}
SPL {X  -150.445, Y  +730.933, Z    +0.000, E1   -71.979, E3 +32239.003}
SPL {X  -147.389, Y  +738.737, Z    +0.000, E1   -71.634, E3 +32247.076}
SPL {X  -144.044, Y  +746.129, Z    +0.000, E1   -71.236, E3 +32255.070}
SPL {X  -140.684, Y  +752.689, Z    +0.000, E1   -70.820, E3 +32262.445}
SPL {X  -137.335, Y  +758.572, Z    +0.000, E1   -70.388, E3 +32269.253}
SPL {X  -133.651, Y  +764.444, Z    +0.000, E1   -69.897, E3 +32276.205}
SPL {X  -129.492, Y  +770.461, Z    +0.000, E1   -69.311, E3 +32283.445}
SPL {X  -125.168, Y  +776.148, Z    +0.000, E1   -68.666, E3 +32290.321}
SPL {X  -122.036, Y  +779.960, Z    +0.000, E1   -68.144, E3 +32294.925}
SPL {X   -80.879, Y  +814.541, Z    +0.000, E1   -55.704, E3 +32416.242}
ENDSPLINE

SPLINE
SPL {X  -125.518, Y  +775.707, Z    +0.000, E1   -52.189, E3 +32587.720}
SPL {X  -144.748, Y  +744.653, Z    +0.000, E1   -45.208, E3 +32605.916}
SPL {X  -153.147, Y  +722.791, Z    +0.000, E1   -36.417, E3 +32612.311}
SPL {X  -158.456, Y  +698.602, Z    +0.000, E1   -21.523, E3 +32616.157}
SPL {X  -159.738, Y  +685.469, Z    +0.000, E1   -10.595, E3 +32617.212}
SPL {X  -159.986, Y  +677.650, Z    +0.000, E1    -3.291, E3 +32617.467}
SPL {X  -159.990, Y  +674.500, Z    +0.000, E1    +0.000, E3 +32617.497}
SPL {X  -159.990, Y  +672.716, Z    +0.000, E1    +3.405, E3 +32617.513}
SPL {X  -159.990, Y  +668.521, Z    +0.000, E1   +13.007, E3 +32617.633}
SPL {X  -159.990, Y  +662.839, Z    +0.000, E1   +26.519, E3 +32617.975}
SPL {X  -159.990, Y  +653.836, Z    +0.000, E1   +43.967, E3 +32618.905}
SPL {X  -159.990, Y  +641.022, Z    +0.000, E1   +57.726, E3 +32621.214}
SPL {X  -159.990, Y  +617.987, Z    +0.000, E1   +67.134, E3 +32627.110}
SPL {X  -159.990, Y  +532.407, Z    +0.000, E1   +73.084, E3 +32658.016}
SPL {X  -159.990, Y  +382.957, Z    +0.000, E1   +73.647, E3 +32734.276}
SPL {X  -159.615, Y  +366.548, Z    +0.000, E1   +73.602, E3 +32744.918}
SPL {X  -157.928, Y  +351.899, Z    +0.000, E1   +73.451, E3 +32755.773}
ENDSPLINE

SPLINE
SPL {X  -159.990, Y  +380.170, Z    +0.000, E1   +69.785, E3 +32771.913}
ENDSPLINE

SPLINE
SPL {X  -158.227, Y  +353.814, Z    +0.000, E1   +70.663, E3 +32783.806}
SPL {X  -155.560, Y  +340.111, Z    +0.000, E1   +70.976, E3 +32790.829}
SPL {X  -151.918, Y  +327.322, Z    +0.000, E1   +71.266, E3 +32797.172}
SPL {X  -144.697, Y  +309.238, Z    +0.000, E1   +71.848, E3 +32804.122}
SPL {X  -140.298, Y  +300.601, Z    +0.000, E1   +71.461, E3 +32812.409}
SPL {X  -135.903, Y  +293.078, Z    +0.000, E1   +70.930, E3 +32820.947}
SPL {X  -132.382, Y  +287.656, Z    +0.000, E1   +70.425, E3 +32827.339}
SPL {X  -128.648, Y  +282.387, Z    +0.000, E1   +69.939, E3 +32833.519}
SPL {X  -125.063, Y  +277.720, Z    +0.000, E1   +69.378, E3 +32839.095}
SPL {X  -122.086, Y  +274.099, Z    +0.000, E1   +68.932, E3 +32843.340}
SPL {X   -84.117, Y  +241.407, Z    +0.000, E1   +58.224, E3 +32934.223}
ENDSPLINE

SPLINE
SPL {X  -116.986, Y  +268.362, Z    +0.000, E1   +53.233, E3 +33128.138}
SPL {X  -146.319, Y  +312.789, Z    +0.000, E1   +44.152, E3 +33158.604}
SPL {X  -155.980, Y  +341.904, Z    +0.000, E1   +30.583, E3 +33165.900}
SPL {X  -159.279, Y  +362.429, Z    +0.000, E1   +16.013, E3 +33168.286}
SPL {X  -159.976, Y  +375.387, Z    +0.000, E1    +4.229, E3 +33168.937}
SPL {X  -159.990, Y  +379.485, Z    +0.000, E1    +0.028, E3 +33168.982}
SPL {X  -159.990, Y  +381.270, Z    +0.000, E1    -3.383, E3 +33168.999}
SPL {X  -159.990, Y  +386.246, Z    +0.000, E1   -14.704, E3 +33169.156}
SPL {X  -159.990, Y  +394.075, Z    +0.000, E1   -32.836, E3 +33169.717}
SPL {X  -159.990, Y  +405.152, Z    +0.000, E1   -50.697, E3 +33171.141}
SPL {X  -159.990, Y  +423.293, Z    +0.000, E1   -63.280, E3 +33175.143}
SPL {X  -159.990, Y  +493.649, Z    +0.000, E1   -71.671, E3 +33200.847}
SPL {X  -159.990, Y  +662.531, Z    +0.000, E1   -73.010, E3 +33287.670}
SPL {X  -159.805, Y  +684.185, Z    +0.000, E1   -72.979, E3 +33301.954}
SPL {X  -158.295, Y  +699.729, Z    +0.000, E1   -72.830, E3 +33313.624}
SPL {X  -155.857, Y  +712.630, Z    +0.000, E1   -72.572, E3 +33324.553}
SPL {X  -153.206, Y  +722.596, Z    +0.000, E1   -72.287, E3 +33333.734}
SPL {X  -150.445, Y  +730.933, Z    +0.000, E1   -71.979, E3 +33341.944}
SPL {X  -147.389, Y  +738.737, Z    +0.000, E1   -71.634, E3 +33350.017}
SPL {X  -144.044, Y  +746.129, Z    +0.000, E1   -71.236, E3 +33358.011}
SPL {X  -140.684, Y  +752.689, Z    +0.000, E1   -70.820, E3 +33365.387}
SPL {X  -137.335, Y  +758.572, Z    +0.000, E1   -70.388, E3 +33372.194}
SPL {X  -133.651, Y  +764.444, Z    +0.000, E1   -69.897, E3 +33379.146}
SPL {X  -129.492, Y  +770.461, Z    +0.000, E1   -69.311, E3 +33386.386}
SPL {X  -125.168, Y  +776.148, Z    +0.000, E1   -68.666, E3 +33393.262}
SPL {X  -122.036, Y  +779.960, Z    +0.000, E1   -68.144, E3 +33397.866}
SPL {X   -80.879, Y  +814.541, Z    +0.000, E1   -55.704, E3 +33519.184}
ENDSPLINE

SPLINE
SPL {X  -125.518, Y  +775.707, Z    +0.000, E1   -52.189, E3 +33690.661}
SPL {X  -144.748, Y  +744.653, Z    +0.000, E1   -45.208, E3 +33708.857}
SPL {X  -153.147, Y  +722.791, Z    +0.000, E1   -36.417, E3 +33715.252}
SPL {X  -157.402, Y  +705.160, Z    +0.000, E1   -26.108, E3 +33718.348}
SPL {X  -159.480, Y  +689.270, Z    +0.000, E1   -14.023, E3 +33719.913}
SPL {X  -159.986, Y  +677.650, Z    +0.000, E1    -3.291, E3 +33720.408}
SPL {X  -159.990, Y  +674.500, Z    +0.000, E1    +0.000, E3 +33720.438}
SPL {X  -159.990, Y  +672.716, Z    +0.000, E1    +3.405, E3 +33720.455}
SPL {X  -159.990, Y  +668.521, Z    +0.000, E1   +13.007, E3 +33720.574}
SPL {X  -159.990, Y  +664.286, Z    +0.000, E1   +23.338, E3 +33720.805}
SPL {X  -159.990, Y  +658.431, Z    +0.000, E1   +35.998, E3 +33721.300}
SPL {X  -159.990, Y  +650.524, Z    +0.000, E1   +48.779, E3 +33722.288}
SPL {X  -159.990, Y  +641.022, Z    +0.000, E1   +57.726, E3 +33724.155}
SPL {X  -159.990, Y  +617.987, Z    +0.000, E1   +67.134, E3 +33730.051}
SPL {X  -159.990, Y  +532.407, Z    +0.000, E1   +73.084, E3 +33760.957}
SPL {X  -159.990, Y  +390.607, Z    +0.000, E1   +73.632, E3 +33832.494}
SPL {X  -159.886, Y  +371.742, Z    +0.000, E1   +73.650, E3 +33844.280}
SPL {X  -157.928, Y  +351.899, Z    +0.000, E1   +73.451, E3 +33858.714}
ENDSPLINE

SPLINE
SPL {X  -159.990, Y  +380.170, Z    +0.000, E1   +69.785, E3 +33874.854}
ENDSPLINE

SPLINE
SPL {X  -158.227, Y  +353.814, Z    +0.000, E1   +70.663, E3 +33886.748}
SPL {X  -155.560, Y  +340.111, Z    +0.000, E1   +70.976, E3 +33893.770}
SPL {X  -151.918, Y  +327.322, Z    +0.000, E1   +71.266, E3 +33900.113}
SPL {X  -144.697, Y  +309.238, Z    +0.000, E1   +71.848, E3 +33907.063}
SPL {X  -140.298, Y  +300.601, Z    +0.000, E1   +71.461, E3 +33915.350}
SPL {X  -137.001, Y  +294.872, Z    +0.000, E1   +71.048, E3 +33921.859}
SPL {X  -133.301, Y  +289.026, Z    +0.000, E1   +70.567, E3 +33928.645}
SPL {X  -129.603, Y  +283.692, Z    +0.000, E1   +70.051, E3 +33934.945}
SPL {X  -125.807, Y  +278.659, Z    +0.000, E1   +69.508, E3 +33940.904}
SPL {X  -122.086, Y  +274.099, Z    +0.000, E1   +68.932, E3 +33946.281}
SPL {X   -84.117, Y  +241.407, Z    +0.000, E1   +58.224, E3 +34037.164}
ENDSPLINE

SPLINE
SPL {X  -116.986, Y  +268.362, Z    +0.000, E1   +53.233, E3 +34231.080}
SPL {X  -146.319, Y  +312.789, Z    +0.000, E1   +44.152, E3 +34261.546}
SPL {X  -157.053, Y  +346.986, Z    +0.000, E1   +27.437, E3 +34269.577}
SPL {X  -159.518, Y  +365.226, Z    +0.000, E1   +13.562, E3 +34271.442}
SPL {X  -159.976, Y  +375.387, Z    +0.000, E1    +4.229, E3 +34271.878}
SPL {X  -159.990, Y  +379.485, Z    +0.000, E1    +0.028, E3 +34271.923}
SPL {X  -159.990, Y  +381.270, Z    +0.000, E1    -3.383, E3 +34271.940}
SPL {X  -159.990, Y  +386.246, Z    +0.000, E1   -14.704, E3 +34272.098}
SPL {X  -159.990, Y  +394.075, Z    +0.000, E1   -32.836, E3 +34272.658}
SPL {X  -159.990, Y  +405.152, Z    +0.000, E1   -50.697, E3 +34274.082}
SPL {X  -159.990, Y  +423.293, Z    +0.000, E1   -63.280, E3 +34278.084}
SPL {X  -159.990, Y  +493.649, Z    +0.000, E1   -71.671, E3 +34303.788}
SPL {X  -159.990, Y  +662.531, Z    +0.000, E1   -73.010, E3 +34390.611}
SPL {X  -159.805, Y  +684.185, Z    +0.000, E1   -72.979, E3 +34404.895}
SPL {X  -158.295, Y  +699.729, Z    +0.000, E1   -72.830, E3 +34416.565}
SPL {X  -155.857, Y  +712.630, Z    +0.000, E1   -72.572, E3 +34427.494}
SPL {X  -153.206, Y  +722.596, Z    +0.000, E1   -72.287, E3 +34436.675}
SPL {X  -150.445, Y  +730.933, Z    +0.000, E1   -71.979, E3 +34444.885}
SPL {X  -147.389, Y  +738.737, Z    +0.000, E1   -71.634, E3 +34452.958}
SPL {X  -144.044, Y  +746.129, Z    +0.000, E1   -71.236, E3 +34460.952}
SPL {X  -140.684, Y  +752.689, Z    +0.000, E1   -70.820, E3 +34468.328}
SPL {X  -136.099, Y  +760.606, Z    +0.000, E1   -70.253, E3 +34477.483}
SPL {X  -131.456, Y  +767.693, Z    +0.000, E1   -69.587, E3 +34485.995}
SPL {X  -128.507, Y  +771.803, Z    +0.000, E1   -69.145, E3 +34490.977}
SPL {X  -125.168, Y  +776.148, Z    +0.000, E1   -68.666, E3 +34496.204}
SPL {X  -122.036, Y  +779.960, Z    +0.000, E1   -68.144, E3 +34500.807}
SPL {X   -80.879, Y  +814.541, Z    +0.000, E1   -55.704, E3 +34622.125}
ENDSPLINE

SPLINE
SPL {X  -125.518, Y  +775.707, Z    +0.000, E1   -52.189, E3 +34793.602}
SPL {X  -150.797, Y  +729.951, Z    +0.000, E1   -39.777, E3 +34816.337}
SPL {X  -158.456, Y  +698.602, Z    +0.000, E1   -21.523, E3 +34822.040}
SPL {X  -159.738, Y  +685.469, Z    +0.000, E1   -10.595, E3 +34823.094}
SPL {X  -159.986, Y  +677.650, Z    +0.000, E1    -3.291, E3 +34823.349}
SPL {X  -159.990, Y  +674.500, Z    +0.000, E1    +0.000, E3 +34823.379}
SPL {X  -159.990, Y  +672.716, Z    +0.000, E1    +3.405, E3 +34823.396}
SPL {X  -159.990, Y  +668.521, Z    +0.000, E1   +13.007, E3 +34823.515}
SPL {X  -159.990, Y  +662.839, Z    +0.000, E1   +26.519, E3 +34823.857}
SPL {X  -159.990, Y  +653.836, Z    +0.000, E1   +43.967, E3 +34824.787}
SPL {X  -159.990, Y  +641.022, Z    +0.000, E1   +57.726, E3 +34827.096}
SPL {X  -159.990, Y  +617.987, Z    +0.000, E1   +67.134, E3 +34832.992}
SPL {X  -159.990, Y  +532.407, Z    +0.000, E1   +73.084, E3 +34863.899}
SPL {X  -159.990, Y  +382.957, Z    +0.000, E1   +73.647, E3 +34940.158}
SPL {X  -159.615, Y  +366.548, Z    +0.000, E1   +73.602, E3 +34950.801}
SPL {X  -157.928, Y  +351.899, Z    +0.000, E1   +73.451, E3 +34961.655}
ENDSPLINE

SPLINE
SPL {X  -159.990, Y  +380.170, Z    +0.000, E1   +69.785, E3 +34977.795}
ENDSPLINE

SPLINE
SPL {X  -158.227, Y  +353.814, Z    +0.000, E1   +70.663, E3 +34989.689}
SPL {X  -155.560, Y  +340.111, Z    +0.000, E1   +70.976, E3 +34996.711}
SPL {X  -151.918, Y  +327.322, Z    +0.000, E1   +71.266, E3 +35003.054}
SPL {X  -144.697, Y  +309.238, Z    +0.000, E1   +71.848, E3 +35010.004}
SPL {X  -140.298, Y  +300.601, Z    +0.000, E1   +71.461, E3 +35018.292}
SPL {X  -137.001, Y  +294.872, Z    +0.000, E1   +71.048, E3 +35024.800}
SPL {X  -133.301, Y  +289.026, Z    +0.000, E1   +70.567, E3 +35031.586}
SPL {X  -128.648, Y  +282.387, Z    +0.000, E1   +69.939, E3 +35039.402}
SPL {X  -125.063, Y  +277.720, Z    +0.000, E1   +69.378, E3 +35044.977}
SPL {X  -122.086, Y  +274.099, Z    +0.000, E1   +68.932, E3 +35049.223}
SPL {X   -84.117, Y  +241.407, Z    +0.000, E1   +58.224, E3 +35140.105}
ENDSPLINE

SPLINE
SPL {X  -106.708, Y  +258.294, Z    +0.000, E1   +53.789, E3 +35318.892}
SPL {X  -137.973, Y  +296.505, Z    +0.000, E1   +48.844, E3 +35357.672}
SPL {X  -154.359, Y  +335.426, Z    +0.000, E1   +34.338, E3 +35370.568}
SPL {X  -159.279, Y  +362.429, Z    +0.000, E1   +16.013, E3 +35374.168}
SPL {X  -159.976, Y  +375.387, Z    +0.000, E1    +4.229, E3 +35374.819}
SPL {X  -159.990, Y  +379.485, Z    +0.000, E1    +0.028, E3 +35374.864}
SPL {X  -159.990, Y  +381.270, Z    +0.000, E1    -3.383, E3 +35374.881}
SPL {X  -159.990, Y  +384.811, Z    +0.000, E1   -11.531, E3 +35374.971}
SPL {X  -159.990, Y  +390.180, Z    +0.000, E1   -24.142, E3 +35375.274}
SPL {X  -159.990, Y  +397.074, Z    +0.000, E1   -39.012, E3 +35375.884}
SPL {X  -159.990, Y  +405.152, Z    +0.000, E1   -50.697, E3 +35377.024}
SPL {X  -159.990, Y  +423.293, Z    +0.000, E1   -63.280, E3 +35381.025}
SPL {X  -159.990, Y  +493.649, Z    +0.000, E1   -71.671, E3 +35406.729}
SPL {X  -159.990, Y  +654.929, Z    +0.000, E1   -72.988, E3 +35488.679}
SPL {X  -159.990, Y  +668.018, Z    +0.000, E1   -72.989, E3 +35497.171}
SPL {X  -159.805, Y  +684.185, Z    +0.000, E1   -72.979, E3 +35507.836}
SPL {X  -158.295, Y  +699.729, Z    +0.000, E1   -72.830, E3 +35519.506}
SPL {X  -155.857, Y  +712.630, Z    +0.000, E1   -72.572, E3 +35530.435}
SPL {X  -153.206, Y  +722.596, Z    +0.000, E1   -72.287, E3 +35539.616}
SPL {X  -150.445, Y  +730.933, Z    +0.000, E1   -71.979, E3 +35547.827}
SPL {X  -147.389, Y  +738.737, Z    +0.000, E1   -71.634, E3 +35555.899}
SPL {X  -144.044, Y  +746.129, Z    +0.000, E1   -71.236, E3 +35563.894}
SPL {X  -140.684, Y  +752.689, Z    +0.000, E1   -70.820, E3 +35571.269}
SPL {X  -136.099, Y  +760.606, Z    +0.000, E1   -70.253, E3 +35580.424}
SPL {X  -131.456, Y  +767.693, Z    +0.000, E1   -69.587, E3 +35588.936}
SPL {X  -128.507, Y  +771.803, Z    +0.000, E1   -69.145, E3 +35593.918}
SPL {X  -125.168, Y  +776.148, Z    +0.000, E1   -68.666, E3 +35599.145}
SPL {X  -122.036, Y  +779.960, Z    +0.000, E1   -68.144, E3 +35603.748}
SPL {X   -80.879, Y  +814.541, Z    +0.000, E1   -55.704, E3 +35725.066}
ENDSPLINE

SPLINE
SPL {X  -125.518, Y  +775.707, Z    +0.000, E1   -52.189, E3 +35896.543}
SPL {X  -150.797, Y  +729.951, Z    +0.000, E1   -39.777, E3 +35919.278}
SPL {X  -157.402, Y  +705.160, Z    +0.000, E1   -26.108, E3 +35924.230}
SPL {X  -159.480, Y  +689.270, Z    +0.000, E1   -14.023, E3 +35925.796}
SPL {X  -159.986, Y  +677.650, Z    +0.000, E1    -3.291, E3 +35926.290}
SPL {X  -159.990, Y  +674.500, Z    +0.000, E1    +0.000, E3 +35926.320}
SPL {X  -159.990, Y  +672.716, Z    +0.000, E1    +3.405, E3 +35926.337}
SPL {X  -159.990, Y  +668.521, Z    +0.000, E1   +13.007, E3 +35926.456}
SPL {X  -159.990, Y  +662.839, Z    +0.000, E1   +26.519, E3 +35926.798}
SPL {X  -159.990, Y  +653.836, Z    +0.000, E1   +43.967, E3 +35927.729}
SPL {X  -159.990, Y  +641.022, Z    +0.000, E1   +57.726, E3 +35930.038}
SPL {X  -159.990, Y  +617.987, Z    +0.000, E1   +67.134, E3 +35935.933}
SPL {X  -159.990, Y  +532.407, Z    +0.000, E1   +73.084, E3 +35966.840}
SPL {X  -159.990, Y  +382.957, Z    +0.000, E1   +73.647, E3 +36043.099}
SPL {X  -159.196, Y  +361.585, Z    +0.000, E1   +73.581, E3 +36057.222}
SPL {X  -157.239, Y  +347.958, Z    +0.000, E1   +73.365, E3 +36067.817}
ENDSPLINE

SPLINE
SPL {X  -159.990, Y  +380.170, Z    +0.000, E1   +69.785, E3 +36080.736}
ENDSPLINE

SPLINE
SPL {X  -158.227, Y  +353.814, Z    +0.000, E1   +70.663, E3 +36092.630}
SPL {X  -155.560, Y  +340.111, Z    +0.000, E1   +70.976, E3 +36099.652}
SPL {X  -151.918, Y  +327.322, Z    +0.000, E1   +71.266, E3 +36105.996}
SPL {X  -144.697, Y  +309.238, Z    +0.000, E1   +71.848, E3 +36112.945}
SPL {X  -140.298, Y  +300.601, Z    +0.000, E1   +71.461, E3 +36121.233}
SPL {X  -137.001, Y  +294.872, Z    +0.000, E1   +71.048, E3 +36127.741}
SPL {X  -133.301, Y  +289.026, Z    +0.000, E1   +70.567, E3 +36134.527}
SPL {X  -129.603, Y  +283.692, Z    +0.000, E1   +70.051, E3 +36140.827}
SPL {X  -125.807, Y  +278.659, Z    +0.000, E1   +69.508, E3 +36146.786}
SPL {X  -122.086, Y  +274.099, Z    +0.000, E1   +68.932, E3 +36152.164}
SPL {X   -84.117, Y  +241.407, Z    +0.000, E1   +58.224, E3 +36243.046}
ENDSPLINE

SPLINE
SPL {X  -106.708, Y  +258.294, Z    +0.000, E1   +53.789, E3 +36421.833}
SPL {X  -137.973, Y  +296.505, Z    +0.000, E1   +48.844, E3 +36460.613}
SPL {X  -154.359, Y  +335.426, Z    +0.000, E1   +34.338, E3 +36473.509}
SPL {X  -159.279, Y  +362.429, Z    +0.000, E1   +16.013, E3 +36477.110}
SPL {X  -159.976, Y  +375.387, Z    +0.000, E1    +4.229, E3 +36477.760}
SPL {X  -159.990, Y  +379.485, Z    +0.000, E1    +0.028, E3 +36477.805}
SPL {X  -159.990, Y  +381.270, Z    +0.000, E1    -3.383, E3 +36477.822}
SPL {X  -159.990, Y  +386.246, Z    +0.000, E1   -14.704, E3 +36477.980}
SPL {X  -159.990, Y  +394.075, Z    +0.000, E1   -32.836, E3 +36478.541}
SPL {X  -159.990, Y  +405.152, Z    +0.000, E1   -50.697, E3 +36479.965}
SPL {X  -159.990, Y  +423.293, Z    +0.000, E1   -63.280, E3 +36483.966}
SPL {X  -159.990, Y  +493.649, Z    +0.000, E1   -71.671, E3 +36509.670}
SPL {X  -159.990, Y  +662.531, Z    +0.000, E1   -73.010, E3 +36596.493}
SPL {X  -159.805, Y  +684.185, Z    +0.000, E1   -72.979, E3 +36610.777}
SPL {X  -158.295, Y  +699.729, Z    +0.000, E1   -72.830, E3 +36622.447}
SPL {X  -155.857, Y  +712.630, Z    +0.000, E1   -72.572, E3 +36633.376}
SPL {X  -153.206, Y  +722.596, Z    +0.000, E1   -72.287, E3 +36642.557}
SPL {X  -150.445, Y  +730.933, Z    +0.000, E1   -71.979, E3 +36650.768}
SPL {X  -147.389, Y  +738.737, Z    +0.000, E1   -71.634, E3 +36658.840}
SPL {X  -144.044, Y  +746.129, Z    +0.000, E1   -71.236, E3 +36666.835}
SPL {X  -140.684, Y  +752.689, Z    +0.000, E1   -70.820, E3 +36674.210}
SPL {X  -136.099, Y  +760.606, Z    +0.000, E1   -70.253, E3 +36683.366}
SPL {X  -131.456, Y  +767.693, Z    +0.000, E1   -69.587, E3 +36691.877}
SPL {X  -127.440, Y  +773.226, Z    +0.000, E1   -69.006, E3 +36698.561}
SPL {X  -123.127, Y  +778.659, Z    +0.000, E1   -68.349, E3 +36705.103}
SPL {X   -80.879, Y  +814.541, Z    +0.000, E1   -55.704, E3 +36828.007}
ENDSPLINE

SPLINE
SPL {X  -125.518, Y  +775.707, Z    +0.000, E1   -52.189, E3 +36999.484}
SPL {X  -144.748, Y  +744.653, Z    +0.000, E1   -45.208, E3 +37017.680}
SPL {X  -153.147, Y  +722.791, Z    +0.000, E1   -36.417, E3 +37024.076}
SPL {X  -157.402, Y  +705.160, Z    +0.000, E1   -26.108, E3 +37027.171}
SPL {X  -159.480, Y  +689.270, Z    +0.000, E1   -14.023, E3 +37028.737}
SPL {X  -159.986, Y  +677.650, Z    +0.000, E1    -3.291, E3 +37029.231}
SPL {X  -159.990, Y  +674.500, Z    +0.000, E1    +0.000, E3 +37029.262}
SPL {X  -159.990, Y  +672.716, Z    +0.000, E1    +3.405, E3 +37029.278}
SPL {X  -159.990, Y  +668.521, Z    +0.000, E1   +13.007, E3 +37029.397}
SPL {X  -159.990, Y  +664.286, Z    +0.000, E1   +23.338, E3 +37029.629}
SPL {X  -159.990, Y  +658.431, Z    +0.000, E1   +35.998, E3 +37030.123}
SPL {X  -159.990, Y  +650.524, Z    +0.000, E1   +48.779, E3 +37031.112}
SPL {X  -159.990, Y  +641.022, Z    +0.000, E1   +57.726, E3 +37032.979}
SPL {X  -159.990, Y  +617.987, Z    +0.000, E1   +67.134, E3 +37038.874}
SPL {X  -159.990, Y  +532.407, Z    +0.000, E1   +73.084, E3 +37069.781}
SPL {X  -159.990, Y  +390.607, Z    +0.000, E1   +73.632, E3 +37141.317}
SPL {X  -159.886, Y  +371.742, Z    +0.000, E1   +73.650, E3 +37153.104}
SPL {X  -157.928, Y  +351.899, Z    +0.000, E1   +73.451, E3 +37167.537}
ENDSPLINE

SPLINE
SPL {X  -159.990, Y  +380.170, Z    +0.000, E1   +69.785, E3 +37183.678}
ENDSPLINE

SPLINE
SPL {X  -158.227, Y  +353.814, Z    +0.000, E1   +70.663, E3 +37195.571}
SPL {X  -155.560, Y  +340.111, Z    +0.000, E1   +70.976, E3 +37202.593}
SPL {X  -151.918, Y  +327.322, Z    +0.000, E1   +71.266, E3 +37208.937}
SPL {X  -144.697, Y  +309.238, Z    +0.000, E1   +71.848, E3 +37215.886}
SPL {X  -140.298, Y  +300.601, Z    +0.000, E1   +71.461, E3 +37224.174}
SPL {X  -135.903, Y  +293.078, Z    +0.000, E1   +70.930, E3 +37232.712}
SPL {X  -132.382, Y  +287.656, Z    +0.000, E1   +70.425, E3 +37239.103}
SPL {X  -128.648, Y  +282.387, Z    +0.000, E1   +69.939, E3 +37245.284}
SPL {X  -125.063, Y  +277.720, Z    +0.000, E1   +69.378, E3 +37250.860}
SPL {X  -122.086, Y  +274.099, Z    +0.000, E1   +68.932, E3 +37255.105}
SPL {X   -84.117, Y  +241.407, Z    +0.000, E1   +58.224, E3 +37345.988}
ENDSPLINE

SPLINE
SPL {X  -106.708, Y  +258.294, Z    +0.000, E1   +53.789, E3 +37524.775}
SPL {X  -137.973, Y  +296.505, Z    +0.000, E1   +48.844, E3 +37563.555}
SPL {X  -154.359, Y  +335.426, Z    +0.000, E1   +34.338, E3 +37576.451}
SPL {X  -159.279, Y  +362.429, Z    +0.000, E1   +16.013, E3 +37580.051}
SPL {X  -159.976, Y  +375.387, Z    +0.000, E1    +4.229, E3 +37580.701}
SPL {X  -159.990, Y  +379.485, Z    +0.000, E1    +0.028, E3 +37580.746}
SPL {X  -159.990, Y  +381.270, Z    +0.000, E1    -3.383, E3 +37580.764}
SPL {X  -159.990, Y  +384.811, Z    +0.000, E1   -11.531, E3 +37580.854}
SPL {X  -159.990, Y  +390.180, Z    +0.000, E1   -24.142, E3 +37581.157}
SPL {X  -159.990, Y  +397.074, Z    +0.000, E1   -39.012, E3 +37581.767}
SPL {X  -159.990, Y  +405.152, Z    +0.000, E1   -50.697, E3 +37582.906}
SPL {X  -159.990, Y  +423.293, Z    +0.000, E1   -63.280, E3 +37586.907}
SPL {X  -159.990, Y  +493.649, Z    +0.000, E1   -71.671, E3 +37612.611}
SPL {X  -159.990, Y  +662.531, Z    +0.000, E1   -73.010, E3 +37699.434}
SPL {X  -159.805, Y  +684.185, Z    +0.000, E1   -72.979, E3 +37713.718}
SPL {X  -158.739, Y  +696.464, Z    +0.000, E1   -72.862, E3 +37722.837}
SPL {X  -156.417, Y  +710.124, Z    +0.000, E1   -72.650, E3 +37734.060}
SPL {X  -153.206, Y  +722.596, Z    +0.000, E1   -72.287, E3 +37745.499}
SPL {X  -150.445, Y  +730.933, Z    +0.000, E1   -71.979, E3 +37753.709}
SPL {X  -147.389, Y  +738.737, Z    +0.000, E1   -71.634, E3 +37761.782}
SPL {X  -144.044, Y  +746.129, Z    +0.000, E1   -71.236, E3 +37769.776}
SPL {X  -140.684, Y  +752.689, Z    +0.000, E1   -70.820, E3 +37777.151}
SPL {X  -137.335, Y  +758.572, Z    +0.000, E1   -70.388, E3 +37783.959}
SPL {X  -134.566, Y  +763.037, Z    +0.000, E1   -70.007, E3 +37789.255}
SPL {X  -131.456, Y  +767.693, Z    +0.000, E1   -69.587, E3 +37794.818}
SPL {X  -127.440, Y  +773.226, Z    +0.000, E1   -69.006, E3 +37801.502}
SPL {X  -123.127, Y  +778.659, Z    +0.000, E1   -68.349, E3 +37808.044}
SPL {X   -80.879, Y  +814.541, Z    +0.000, E1   -55.704, E3 +37930.948}
ENDSPLINE

SPLINE
SPL {X  -125.518, Y  +775.707, Z    +0.000, E1   -52.189, E3 +38102.426}
SPL {X  -144.748, Y  +744.653, Z    +0.000, E1   -45.208, E3 +38120.621}
SPL {X  -153.147, Y  +722.791, Z    +0.000, E1   -36.417, E3 +38127.017}
SPL {X  -157.402, Y  +705.160, Z    +0.000, E1   -26.108, E3 +38130.112}
SPL {X  -159.480, Y  +689.270, Z    +0.000, E1   -14.023, E3 +38131.678}
SPL {X  -159.986, Y  +677.650, Z    +0.000, E1    -3.291, E3 +38132.172}
SPL {X  -159.990, Y  +674.500, Z    +0.000, E1    +0.000, E3 +38132.203}
SPL {X  -159.990, Y  +672.716, Z    +0.000, E1    +3.405, E3 +38132.219}
SPL {X  -159.990, Y  +668.521, Z    +0.000, E1   +13.007, E3 +38132.338}
SPL {X  -159.990, Y  +662.839, Z    +0.000, E1   +26.519, E3 +38132.681}
SPL {X  -159.990, Y  +653.836, Z    +0.000, E1   +43.967, E3 +38133.611}
SPL {X  -159.990, Y  +641.022, Z    +0.000, E1   +57.726, E3 +38135.920}
SPL {X  -159.990, Y  +617.987, Z    +0.000, E1   +67.134, E3 +38141.815}
SPL {X  -159.990, Y  +532.407, Z    +0.000, E1   +73.084, E3 +38172.722}
SPL {X  -159.990, Y  +382.957, Z    +0.000, E1   +73.647, E3 +38248.982}
SPL {X  -159.615, Y  +366.548, Z    +0.000, E1   +73.602, E3 +38259.624}
SPL {X  -157.928, Y  +351.899, Z    +0.000, E1   +73.451, E3 +38270.479}
ENDSPLINE

SPLINE
SPL {X  -159.990, Y  +380.170, Z    +0.000, E1   +69.785, E3 +38286.619}
ENDSPLINE

SPLINE
SPL {X  -158.227, Y  +353.814, Z    +0.000, E1   +70.663, E3 +38298.512}
SPL {X  -155.560, Y  +340.111, Z    +0.000, E1   +70.976, E3 +38305.534}
SPL {X  -151.918, Y  +327.322, Z    +0.000, E1   +71.266, E3 +38311.878}
SPL {X  -144.697, Y  +309.238, Z    +0.000, E1   +71.848, E3 +38318.828}
SPL {X  -140.298, Y  +300.601, Z    +0.000, E1   +71.461, E3 +38327.115}
SPL {X  -135.903, Y  +293.078, Z    +0.000, E1   +70.930, E3 +38335.653}
SPL {X  -130.487, Y  +284.926, Z    +0.000, E1   +70.202, E3 +38345.212}
SPL {X  -125.807, Y  +278.659, Z    +0.000, E1   +69.508, E3 +38352.669}
SPL {X  -122.967, Y  +275.148, Z    +0.000, E1   +69.053, E3 +38356.837}
SPL {X  -121.236, Y  +273.103, Z    +0.000, E1   +68.779, E3 +38359.223}
SPL {X   -84.117, Y  +241.407, Z    +0.000, E1   +58.224, E3 +38448.929}
ENDSPLINE

SPLINE
SPL {X  -106.708, Y  +258.294, Z    +0.000, E1   +53.789, E3 +38627.716}
SPL {X  -137.973, Y  +296.505, Z    +0.000, E1   +48.844, E3 +38666.496}
SPL {X  -150.692, Y  +323.752, Z    +0.000, E1   +39.895, E3 +38676.862}
SPL {X  -157.053, Y  +346.986, Z    +0.000, E1   +27.437, E3 +38681.342}
SPL {X  -159.518, Y  +365.226, Z    +0.000, E1   +13.562, E3 +38683.207}
SPL {X  -159.976, Y  +375.387, Z    +0.000, E1    +4.229, E3 +38683.643}
SPL {X  -159.990, Y  +379.485, Z    +0.000, E1    +0.028, E3 +38683.688}
SPL {X  -159.990, Y  +381.270, Z    +0.000, E1    -3.383, E3 +38683.705}
SPL {X  -159.990, Y  +384.811, Z    +0.000, E1   -11.531, E3 +38683.795}
SPL {X  -159.990, Y  +390.180, Z    +0.000, E1   -24.142, E3 +38684.098}
SPL {X  -159.990, Y  +397.074, Z    +0.000, E1   -39.012, E3 +38684.708}
SPL {X  -159.990, Y  +405.152, Z    +0.000, E1   -50.697, E3 +38685.847}
SPL {X  -159.990, Y  +423.293, Z    +0.000, E1   -63.280, E3 +38689.849}
SPL {X  -159.990, Y  +493.649, Z    +0.000, E1   -71.671, E3 +38715.552}
SPL {X  -159.990, Y  +662.531, Z    +0.000, E1   -73.010, E3 +38802.376}
SPL {X  -159.805, Y  +684.185, Z    +0.000, E1   -72.979, E3 +38816.660}
SPL {X  -158.295, Y  +699.729, Z    +0.000, E1   -72.830, E3 +38828.330}
SPL {X  -155.857, Y  +712.630, Z    +0.000, E1   -72.572, E3 +38839.259}
SPL {X  -153.206, Y  +722.596, Z    +0.000, E1   -72.287, E3 +38848.440}
SPL {X  -150.445, Y  +730.933, Z    +0.000, E1   -71.979, E3 +38856.650}
SPL {X  -147.389, Y  +738.737, Z    +0.000, E1   -71.634, E3 +38864.723}
SPL {X  -144.044, Y  +746.129, Z    +0.000, E1   -71.236, E3 +38872.717}
SPL {X  -140.684, Y  +752.689, Z    +0.000, E1   -70.820, E3 +38880.092}
SPL {X  -136.099, Y  +760.606, Z    +0.000, E1   -70.253, E3 +38889.248}
SPL {X  -131.456, Y  +767.693, Z    +0.000, E1   -69.587, E3 +38897.760}
SPL {X  -127.440, Y  +773.226, Z    +0.000, E1   -69.006, E3 +38904.443}
SPL {X  -123.127, Y  +778.659, Z    +0.000, E1   -68.349, E3 +38910.985}
SPL {X   -80.879, Y  +814.541, Z    +0.000, E1   -55.704, E3 +39033.889}
ENDSPLINE

SPLINE
SPL {X  -125.518, Y  +775.707, Z    +0.000, E1   -52.189, E3 +39205.367}
SPL {X  -150.797, Y  +729.951, Z    +0.000, E1   -39.777, E3 +39228.102}
SPL {X  -157.402, Y  +705.160, Z    +0.000, E1   -26.108, E3 +39233.054}
SPL {X  -159.480, Y  +689.270, Z    +0.000, E1   -14.023, E3 +39234.619}
SPL {X  -159.986, Y  +677.650, Z    +0.000, E1    -3.291, E3 +39235.114}
SPL {X  -159.990, Y  +674.500, Z    +0.000, E1    +0.000, E3 +39235.144}
SPL {X  -159.990, Y  +672.716, Z    +0.000, E1    +3.405, E3 +39235.161}
SPL {X  -159.990, Y  +668.521, Z    +0.000, E1   +13.007, E3 +39235.280}
SPL {X  -159.990, Y  +662.839, Z    +0.000, E1   +26.519, E3 +39235.622}
SPL {X  -159.990, Y  +653.836, Z    +0.000, E1   +43.967, E3 +39236.552}
SPL {X  -159.990, Y  +641.022, Z    +0.000, E1   +57.726, E3 +39238.861}
SPL {X  -159.990, Y  +617.987, Z    +0.000, E1   +67.134, E3 +39244.757}
SPL {X  -159.990, Y  +532.407, Z    +0.000, E1   +73.084, E3 +39275.663}
SPL {X  -159.990, Y  +390.607, Z    +0.000, E1   +73.632, E3 +39347.199}
SPL {X  -159.886, Y  +371.742, Z    +0.000, E1   +73.650, E3 +39358.986}
SPL {X  -157.928, Y  +351.899, Z    +0.000, E1   +73.451, E3 +39373.420}
ENDSPLINE

SPLINE
SPL {X  -159.990, Y  +380.170, Z    +0.000, E1   +69.785, E3 +39389.560}
ENDSPLINE

SPLINE
SPL {X  -158.227, Y  +353.814, Z    +0.000, E1   +70.663, E3 +39401.454}
SPL {X  -155.560, Y  +340.111, Z    +0.000, E1   +70.976, E3 +39408.476}
SPL {X  -151.918, Y  +327.322, Z    +0.000, E1   +71.266, E3 +39414.819}
SPL {X  -144.697, Y  +309.238, Z    +0.000, E1   +71.848, E3 +39421.769}
SPL {X  -140.298, Y  +300.601, Z    +0.000, E1   +71.461, E3 +39430.056}
SPL {X  -135.903, Y  +293.078, Z    +0.000, E1   +70.930, E3 +39438.594}
SPL {X  -130.487, Y  +284.926, Z    +0.000, E1   +70.202, E3 +39448.153}
SPL {X  -125.807, Y  +278.659, Z    +0.000, E1   +69.508, E3 +39455.610}
SPL {X  -122.967, Y  +275.148, Z    +0.000, E1   +69.053, E3 +39459.779}
SPL {X  -121.236, Y  +273.103, Z    +0.000, E1   +68.779, E3 +39462.164}
SPL {X   -84.117, Y  +241.407, Z    +0.000, E1   +58.224, E3 +39551.870}
ENDSPLINE

SPLINE
SPL {X  -116.986, Y  +268.362, Z    +0.000, E1   +53.233, E3 +39745.785}
SPL {X  -146.319, Y  +312.789, Z    +0.000, E1   +44.152, E3 +39776.252}
SPL {X  -157.053, Y  +346.986, Z    +0.000, E1   +27.437, E3 +39784.283}
SPL {X  -159.518, Y  +365.226, Z    +0.000, E1   +13.562, E3 +39786.148}
SPL {X  -159.976, Y  +375.387, Z    +0.000, E1    +4.229, E3 +39786.584}
SPL {X  -159.990, Y  +379.485, Z    +0.000, E1    +0.028, E3 +39786.629}
SPL {X  -159.990, Y  +381.270, Z    +0.000, E1    -3.383, E3 +39786.646}
SPL {X  -159.990, Y  +386.246, Z    +0.000, E1   -14.704, E3 +39786.803}
SPL {X  -159.990, Y  +394.075, Z    +0.000, E1   -32.836, E3 +39787.364}
SPL {X  -159.990, Y  +405.152, Z    +0.000, E1   -50.697, E3 +39788.788}
SPL {X  -159.990, Y  +423.293, Z    +0.000, E1   -63.280, E3 +39792.790}
SPL {X  -159.990, Y  +493.649, Z    +0.000, E1   -71.671, E3 +39818.494}
SPL {X  -159.990, Y  +662.531, Z    +0.000, E1   -73.010, E3 +39905.317}
SPL {X  -159.805, Y  +684.185, Z    +0.000, E1   -72.979, E3 +39919.601}
SPL {X  -158.295, Y  +699.729, Z    +0.000, E1   -72.830, E3 +39931.271}
SPL {X  -155.857, Y  +712.630, Z    +0.000, E1   -72.572, E3 +39942.200}
SPL {X  -153.206, Y  +722.596, Z    +0.000, E1   -72.287, E3 +39951.381}
SPL {X  -150.445, Y  +730.933, Z    +0.000, E1   -71.979, E3 +39959.591}
SPL {X  -147.389, Y  +738.737, Z    +0.000, E1   -71.634, E3 +39967.664}
SPL {X  -144.044, Y  +746.129, Z    +0.000, E1   -71.236, E3 +39975.658}
SPL {X  -140.684, Y  +752.689, Z    +0.000, E1   -70.820, E3 +39983.034}
SPL {X  -136.099, Y  +760.606, Z    +0.000, E1   -70.253, E3 +39992.189}
SPL {X  -131.456, Y  +767.693, Z    +0.000, E1   -69.587, E3 +40000.701}
SPL {X  -127.440, Y  +773.226, Z    +0.000, E1   -69.006, E3 +40007.385}
SPL {X  -123.127, Y  +778.659, Z    +0.000, E1   -68.349, E3 +40013.927}
SPL {X   -80.879, Y  +814.541, Z    +0.000, E1   -55.704, E3 +40136.831}
ENDSPLINE

SPLINE
SPL {X  -125.518, Y  +775.707, Z    +0.000, E1   -52.189, E3 +40308.308}
SPL {X  -150.797, Y  +729.951, Z    +0.000, E1   -39.777, E3 +40331.043}
SPL {X  -158.456, Y  +698.602, Z    +0.000, E1   -21.523, E3 +40336.746}
SPL {X  -159.738, Y  +685.469, Z    +0.000, E1   -10.595, E3 +40337.800}
SPL {X  -159.986, Y  +677.650, Z    +0.000, E1    -3.291, E3 +40338.055}
SPL {X  -159.990, Y  +674.500, Z    +0.000, E1    +0.000, E3 +40338.085}
SPL {X  -159.990, Y  +672.716, Z    +0.000, E1    +3.405, E3 +40338.102}
SPL {X  -159.990, Y  +668.521, Z    +0.000, E1   +13.007, E3 +40338.221}
SPL {X  -159.990, Y  +662.839, Z    +0.000, E1   +26.519, E3 +40338.563}
SPL {X  -159.990, Y  +653.836, Z    +0.000, E1   +43.967, E3 +40339.493}
SPL {X  -159.990, Y  +641.022, Z    +0.000, E1   +57.726, E3 +40341.802}
SPL {X  -159.990, Y  +617.987, Z    +0.000, E1   +67.134, E3 +40347.698}
SPL {X  -159.990, Y  +532.407, Z    +0.000, E1   +73.084, E3 +40378.605}
SPL {X  -159.990, Y  +382.957, Z    +0.000, E1   +73.647, E3 +40454.864}
SPL {X  -159.615, Y  +366.548, Z    +0.000, E1   +73.602, E3 +40465.507}
SPL {X  -157.928, Y  +351.899, Z    +0.000, E1   +73.451, E3 +40476.361}
ENDSPLINE

SPLINE
SPL {X  -159.990, Y  +380.170, Z    +0.000, E1   +69.785, E3 +40492.501}
ENDSPLINE

SPLINE
SPL {X  -158.227, Y  +353.814, Z    +0.000, E1   +70.663, E3 +40504.395}
SPL {X  -154.257, Y  +335.055, Z    +0.000, E1   +71.089, E3 +40514.023}
SPL {X  -148.153, Y  +317.104, Z    +0.000, E1   +71.658, E3 +40521.168}
SPL {X  -143.479, Y  +306.716, Z    +0.000, E1   +71.847, E3 +40526.242}
SPL {X  -140.298, Y  +300.601, Z    +0.000, E1   +71.461, E3 +40532.997}
SPL {X  -137.001, Y  +294.872, Z    +0.000, E1   +71.048, E3 +40539.506}
SPL {X  -133.301, Y  +289.026, Z    +0.000, E1   +70.567, E3 +40546.292}
SPL {X  -129.603, Y  +283.692, Z    +0.000, E1   +70.051, E3 +40552.592}
SPL {X  -125.807, Y  +278.659, Z    +0.000, E1   +69.508, E3 +40558.551}
SPL {X  -122.086, Y  +274.099, Z    +0.000, E1   +68.932, E3 +40563.928}
SPL {X   -84.117, Y  +241.407, Z    +0.000, E1   +58.224, E3 +40654.811}
ENDSPLINE

SPLINE
SPL {X  -116.986, Y  +268.362, Z    +0.000, E1   +53.233, E3 +40848.727}
SPL {X  -146.319, Y  +312.789, Z    +0.000, E1   +44.152, E3 +40879.193}
SPL {X  -157.053, Y  +346.986, Z    +0.000, E1   +27.437, E3 +40887.224}
SPL {X  -159.518, Y  +365.226, Z    +0.000, E1   +13.562, E3 +40889.089}
SPL {X  -159.976, Y  +375.387, Z    +0.000, E1    +4.229, E3 +40889.525}
SPL {X  -159.990, Y  +379.485, Z    +0.000, E1    +0.028, E3 +40889.570}
SPL {X  -159.990, Y  +381.270, Z    +0.000, E1    -3.383, E3 +40889.587}
SPL {X  -159.990, Y  +386.246, Z    +0.000, E1   -14.704, E3 +40889.745}
SPL {X  -159.990, Y  +394.075, Z    +0.000, E1   -32.836, E3 +40890.305}
SPL {X  -159.990, Y  +405.152, Z    +0.000, E1   -50.697, E3 +40891.730}
SPL {X  -159.990, Y  +423.293, Z    +0.000, E1   -63.280, E3 +40895.731}
SPL {X  -159.990, Y  +493.649, Z    +0.000, E1   -71.671, E3 +40921.435}
SPL {X  -159.990, Y  +662.531, Z    +0.000, E1   -73.010, E3 +41008.258}
SPL {X  -159.805, Y  +684.185, Z    +0.000, E1   -72.979, E3 +41022.542}
SPL {X  -158.295, Y  +699.729, Z    +0.000, E1   -72.830, E3 +41034.212}
SPL {X  -155.857, Y  +712.630, Z    +0.000, E1   -72.572, E3 +41045.141}
SPL {X  -153.206, Y  +722.596, Z    +0.000, E1   -72.287, E3 +41054.322}
SPL {X  -150.445, Y  +730.933, Z    +0.000, E1   -71.979, E3 +41062.532}
SPL {X  -147.389, Y  +738.737, Z    +0.000, E1   -71.634, E3 +41070.605}
SPL {X  -144.044, Y  +746.129, Z    +0.000, E1   -71.236, E3 +41078.600}
SPL {X  -140.684, Y  +752.689, Z    +0.000, E1   -70.820, E3 +41085.975}
SPL {X  -137.335, Y  +758.572, Z    +0.000, E1   -70.388, E3 +41092.782}
SPL {X  -133.651, Y  +764.444, Z    +0.000, E1   -69.897, E3 +41099.734}
SPL {X  -129.492, Y  +770.461, Z    +0.000, E1   -69.311, E3 +41106.974}
SPL {X  -125.168, Y  +776.148, Z    +0.000, E1   -68.666, E3 +41113.851}
SPL {X  -122.036, Y  +779.960, Z    +0.000, E1   -68.144, E3 +41118.454}
SPL {X   -80.879, Y  +814.541, Z    +0.000, E1   -55.704, E3 +41239.772}
ENDSPLINE

SPLINE
SPL {X  -125.518, Y  +775.707, Z    +0.000, E1   -52.189, E3 +41411.249}
SPL {X  -144.748, Y  +744.653, Z    +0.000, E1   -45.208, E3 +41429.445}
SPL {X  -153.147, Y  +722.791, Z    +0.000, E1   -36.417, E3 +41435.841}
SPL {X  -157.402, Y  +705.160, Z    +0.000, E1   -26.108, E3 +41438.936}
SPL {X  -159.480, Y  +689.270, Z    +0.000, E1   -14.023, E3 +41440.502}
SPL {X  -159.986, Y  +677.650, Z    +0.000, E1    -3.291, E3 +41440.996}
SPL {X  -159.990, Y  +674.500, Z    +0.000, E1    +0.000, E3 +41441.026}
SPL {X  -159.990, Y  +672.716, Z    +0.000, E1    +3.405, E3 +41441.043}
SPL {X  -159.990, Y  +668.521, Z    +0.000, E1   +13.007, E3 +41441.162}
SPL {X  -159.990, Y  +664.286, Z    +0.000, E1   +23.338, E3 +41441.393}
SPL {X  -159.990, Y  +658.431, Z    +0.000, E1   +35.998, E3 +41441.888}
SPL {X  -159.990, Y  +650.524, Z    +0.000, E1   +48.779, E3 +41442.877}
SPL {X  -159.990, Y  +641.022, Z    +0.000, E1   +57.726, E3 +41444.743}
SPL {X  -159.990, Y  +617.987, Z    +0.000, E1   +67.134, E3 +41450.639}
SPL {X  -159.990, Y  +532.407, Z    +0.000, E1   +73.084, E3 +41481.546}
SPL {X  -159.990, Y  +390.607, Z    +0.000, E1   +73.632, E3 +41553.082}
SPL {X  -159.886, Y  +371.742, Z    +0.000, E1   +73.650, E3 +41564.869}
SPL {X  -157.928, Y  +351.899, Z    +0.000, E1   +73.451, E3 +41579.302}
ENDSPLINE

SPLINE
SPL {X  -159.990, Y  +380.170, Z    +0.000, E1   +69.785, E3 +41595.442}
ENDSPLINE

SPLINE
SPL {X  -158.227, Y  +353.814, Z    +0.000, E1   +70.663, E3 +41607.336}
SPL {X  -155.560, Y  +340.111, Z    +0.000, E1   +70.976, E3 +41614.358}
SPL {X  -151.918, Y  +327.322, Z    +0.000, E1   +71.266, E3 +41620.702}
SPL {X  -144.697, Y  +309.238, Z    +0.000, E1   +71.848, E3 +41627.651}
SPL {X  -140.298, Y  +300.601, Z    +0.000, E1   +71.461, E3 +41635.939}
SPL {X  -135.903, Y  +293.078, Z    +0.000, E1   +70.930, E3 +41644.476}
SPL {X  -132.382, Y  +287.656, Z    +0.000, E1   +70.425, E3 +41650.868}
SPL {X  -128.648, Y  +282.387, Z    +0.000, E1   +69.939, E3 +41657.049}
SPL {X  -125.063, Y  +277.720, Z    +0.000, E1   +69.378, E3 +41662.624}
SPL {X  -122.086, Y  +274.099, Z    +0.000, E1   +68.932, E3 +41666.870}
SPL {X   -84.117, Y  +241.407, Z    +0.000, E1   +58.224, E3 +41757.752}
ENDSPLINE

SPLINE
SPL {X  -106.708, Y  +258.294, Z    +0.000, E1   +53.789, E3 +41936.539}
SPL {X  -137.973, Y  +296.505, Z    +0.000, E1   +48.844, E3 +41975.319}
SPL {X  -154.359, Y  +335.426, Z    +0.000, E1   +34.338, E3 +41988.215}
SPL {X  -159.279, Y  +362.429, Z    +0.000, E1   +16.013, E3 +41991.815}
SPL {X  -159.976, Y  +375.387, Z    +0.000, E1    +4.229, E3 +41992.466}
SPL {X  -159.990, Y  +379.485, Z    +0.000, E1    +0.028, E3 +41992.511}
SPL {X  -159.990, Y  +381.270, Z    +0.000, E1    -3.383, E3 +41992.528}
SPL {X  -159.990, Y  +386.246, Z    +0.000, E1   -14.704, E3 +41992.686}
SPL {X  -159.990, Y  +394.075, Z    +0.000, E1   -32.836, E3 +41993.246}
SPL {X  -159.990, Y  +405.152, Z    +0.000, E1   -50.697, E3 +41994.671}
SPL {X  -159.990, Y  +423.293, Z    +0.000, E1   -63.280, E3 +41998.672}
SPL {X  -159.990, Y  +493.649, Z    +0.000, E1   -71.671, E3 +42024.376}
SPL {X  -159.990, Y  +662.531, Z    +0.000, E1   -73.010, E3 +42111.199}
SPL {X  -159.805, Y  +684.185, Z    +0.000, E1   -72.979, E3 +42125.483}
SPL {X  -158.739, Y  +696.464, Z    +0.000, E1   -72.862, E3 +42134.602}
SPL {X  -156.417, Y  +710.124, Z    +0.000, E1   -72.650, E3 +42145.825}
SPL {X  -153.206, Y  +722.596, Z    +0.000, E1   -72.287, E3 +42157.263}
SPL {X  -150.445, Y  +730.933, Z    +0.000, E1   -71.979, E3 +42165.474}
SPL {X  -147.389, Y  +738.737, Z    +0.000, E1   -71.634, E3 +42173.546}
SPL {X  -144.044, Y  +746.129, Z    +0.000, E1   -71.236, E3 +42181.541}
SPL {X  -140.684, Y  +752.689, Z    +0.000, E1   -70.820, E3 +42188.916}
SPL {X  -136.099, Y  +760.606, Z    +0.000, E1   -70.253, E3 +42198.071}
SPL {X  -131.456, Y  +767.693, Z    +0.000, E1   -69.587, E3 +42206.583}
SPL {X  -127.440, Y  +773.226, Z    +0.000, E1   -69.006, E3 +42213.267}
SPL {X  -123.127, Y  +778.659, Z    +0.000, E1   -68.349, E3 +42219.809}
SPL {X   -80.879, Y  +814.541, Z    +0.000, E1   -55.704, E3 +42342.713}
ENDSPLINE

SPLINE
SPL {X  -125.518, Y  +775.707, Z    +0.000, E1   -52.189, E3 +42514.190}
SPL {X  -144.748, Y  +744.653, Z    +0.000, E1   -45.208, E3 +42532.386}
SPL {X  -153.147, Y  +722.791, Z    +0.000, E1   -36.417, E3 +42538.782}
SPL {X  -158.456, Y  +698.602, Z    +0.000, E1   -21.523, E3 +42542.628}
SPL {X  -159.738, Y  +685.469, Z    +0.000, E1   -10.595, E3 +42543.682}
SPL {X  -159.986, Y  +677.650, Z    +0.000, E1    -3.291, E3 +42543.937}
SPL {X  -159.990, Y  +674.500, Z    +0.000, E1    +0.000, E3 +42543.968}
SPL {X  -159.990, Y  +672.716, Z    +0.000, E1    +3.405, E3 +42543.984}
SPL {X  -159.990, Y  +668.521, Z    +0.000, E1   +13.007, E3 +42544.103}
SPL {X  -159.990, Y  +662.839, Z    +0.000, E1   +26.519, E3 +42544.445}
SPL {X  -159.990, Y  +653.836, Z    +0.000, E1   +43.967, E3 +42545.376}
SPL {X  -159.990, Y  +641.022, Z    +0.000, E1   +57.726, E3 +42547.685}
SPL {X  -159.990, Y  +617.987, Z    +0.000, E1   +67.134, E3 +42553.580}
SPL {X  -159.990, Y  +532.407, Z    +0.000, E1   +73.084, E3 +42584.487}
SPL {X  -159.990, Y  +390.607, Z    +0.000, E1   +73.632, E3 +42656.023}
SPL {X  -159.886, Y  +371.742, Z    +0.000, E1   +73.650, E3 +42667.810}
SPL {X  -157.928, Y  +351.899, Z    +0.000, E1   +73.451, E3 +42682.243}
ENDSPLINE

SPLINE
SPL {X  -159.990, Y  +387.996, Z    +0.000, E1   +69.509, E3 +42694.673}
ENDSPLINE

SPLINE
SPL {X  -159.889, Y  +371.819, Z    +0.000, E1   +70.046, E3 +42702.400}
SPL {X  -158.227, Y  +353.814, Z    +0.000, E1   +70.663, E3 +42710.277}
SPL {X  -154.257, Y  +335.055, Z    +0.000, E1   +71.089, E3 +42719.905}
SPL {X  -148.153, Y  +317.104, Z    +0.000, E1   +71.658, E3 +42727.051}
SPL {X  -143.479, Y  +306.716, Z    +0.000, E1   +71.847, E3 +42732.124}
SPL {X  -140.298, Y  +300.601, Z    +0.000, E1   +71.461, E3 +42738.880}
SPL {X  -135.903, Y  +293.078, Z    +0.000, E1   +70.930, E3 +42747.417}
SPL {X  -130.487, Y  +284.926, Z    +0.000, E1   +70.202, E3 +42756.977}
SPL {X  -125.807, Y  +278.659, Z    +0.000, E1   +69.508, E3 +42764.433}
SPL {X  -122.967, Y  +275.148, Z    +0.000, E1   +69.053, E3 +42768.602}
SPL {X  -121.236, Y  +273.103, Z    +0.000, E1   +68.779, E3 +42770.988}
SPL {X   -84.117, Y  +241.407, Z    +0.000, E1   +58.224, E3 +42860.693}
ENDSPLINE

SPLINE
SPL {X  -116.986, Y  +268.362, Z    +0.000, E1   +53.233, E3 +43054.609}
SPL {X  -146.319, Y  +312.789, Z    +0.000, E1   +44.152, E3 +43085.075}
SPL {X  -157.053, Y  +346.986, Z    +0.000, E1   +27.437, E3 +43093.106}
SPL {X  -159.518, Y  +365.226, Z    +0.000, E1   +13.562, E3 +43094.972}
SPL {X  -159.976, Y  +375.387, Z    +0.000, E1    +4.229, E3 +43095.407}
SPL {X  -159.990, Y  +379.485, Z    +0.000, E1    +0.028, E3 +43095.452}
SPL {X  -159.990, Y  +381.270, Z    +0.000, E1    -3.383, E3 +43095.469}
SPL {X  -159.990, Y  +384.811, Z    +0.000, E1   -11.531, E3 +43095.560}
SPL {X  -159.990, Y  +388.002, Z    +0.000, E1   -19.281, E3 +43095.709}
SPL {X  -159.990, Y  +394.075, Z    +0.000, E1   -32.836, E3 +43096.188}
SPL {X  -159.990, Y  +405.152, Z    +0.000, E1   -50.697, E3 +43097.612}
SPL {X  -159.990, Y  +423.293, Z    +0.000, E1   -63.280, E3 +43101.613}
SPL {X  -159.990, Y  +493.649, Z    +0.000, E1   -71.671, E3 +43127.317}
SPL {X  -159.990, Y  +654.929, Z    +0.000, E1   -72.988, E3 +43209.267}
SPL {X  -159.990, Y  +668.018, Z    +0.000, E1   -72.989, E3 +43217.760}
SPL {X  -159.805, Y  +684.185, Z    +0.000, E1   -72.979, E3 +43228.424}
SPL {X  -158.295, Y  +699.729, Z    +0.000, E1   -72.830, E3 +43240.095}
SPL {X  -155.857, Y  +712.630, Z    +0.000, E1   -72.572, E3 +43251.024}
SPL {X  -153.206, Y  +722.596, Z    +0.000, E1   -72.287, E3 +43260.204}
SPL {X  -150.445, Y  +730.933, Z    +0.000, E1   -71.979, E3 +43268.415}
SPL {X  -147.389, Y  +738.737, Z    +0.000, E1   -71.634, E3 +43276.487}
SPL {X  -144.044, Y  +746.129, Z    +0.000, E1   -71.236, E3 +43284.482}
SPL {X  -140.684, Y  +752.689, Z    +0.000, E1   -70.820, E3 +43291.857}
SPL {X  -136.099, Y  +760.606, Z    +0.000, E1   -70.253, E3 +43301.013}
SPL {X  -131.456, Y  +767.693, Z    +0.000, E1   -69.587, E3 +43309.524}
SPL {X  -128.507, Y  +771.803, Z    +0.000, E1   -69.145, E3 +43314.506}
SPL {X  -125.168, Y  +776.148, Z    +0.000, E1   -68.666, E3 +43319.733}
SPL {X  -122.036, Y  +779.960, Z    +0.000, E1   -68.144, E3 +43324.336}
SPL {X   -80.879, Y  +814.541, Z    +0.000, E1   -55.704, E3 +43445.654}
ENDSPLINE

SPLINE
SPL {X  -125.518, Y  +775.707, Z    +0.000, E1   -52.189, E3 +43617.132}
SPL {X  -144.748, Y  +744.653, Z    +0.000, E1   -45.208, E3 +43635.327}
SPL {X  -153.147, Y  +722.791, Z    +0.000, E1   -36.417, E3 +43641.723}
SPL {X  -158.456, Y  +698.602, Z    +0.000, E1   -21.523, E3 +43645.569}
SPL {X  -159.738, Y  +685.469, Z    +0.000, E1   -10.595, E3 +43646.623}
SPL {X  -159.986, Y  +677.650, Z    +0.000, E1    -3.291, E3 +43646.878}
SPL {X  -159.990, Y  +674.500, Z    +0.000, E1    +0.000, E3 +43646.909}
SPL {X  -159.990, Y  +672.716, Z    +0.000, E1    +3.405, E3 +43646.925}
SPL {X  -159.990, Y  +668.521, Z    +0.000, E1   +13.007, E3 +43647.044}
SPL {X  -159.990, Y  +664.286, Z    +0.000, E1   +23.338, E3 +43647.276}
SPL {X  -159.990, Y  +658.431, Z    +0.000, E1   +35.998, E3 +43647.770}
SPL {X  -159.990, Y  +650.524, Z    +0.000, E1   +48.779, E3 +43648.759}
SPL {X  -159.990, Y  +641.022, Z    +0.000, E1   +57.726, E3 +43650.626}
SPL {X  -159.990, Y  +617.987, Z    +0.000, E1   +67.134, E3 +43656.521}
SPL {X  -159.990, Y  +532.407, Z    +0.000, E1   +73.084, E3 +43687.428}
SPL {X  -159.990, Y  +382.957, Z    +0.000, E1   +73.647, E3 +43763.688}
SPL {X  -159.615, Y  +366.548, Z    +0.000, E1   +73.602, E3 +43774.330}
SPL {X  -157.928, Y  +351.899, Z    +0.000, E1   +73.451, E3 +43785.184}
ENDSPLINE

SPLINE
SPL {X  -159.990, Y  +380.170, Z    +0.000, E1   +69.785, E3 +43801.325}
ENDSPLINE

SPLINE
SPL {X  -158.227, Y  +353.814, Z    +0.000, E1   +70.663, E3 +43813.218}
SPL {X  -155.560, Y  +340.111, Z    +0.000, E1   +70.976, E3 +43820.240}
SPL {X  -151.918, Y  +327.322, Z    +0.000, E1   +71.266, E3 +43826.584}
SPL {X  -144.697, Y  +309.238, Z    +0.000, E1   +71.848, E3 +43833.533}
SPL {X  -140.298, Y  +300.601, Z    +0.000, E1   +71.461, E3 +43841.821}
SPL {X  -137.001, Y  +294.872, Z    +0.000, E1   +71.048, E3 +43848.329}
SPL {X  -133.301, Y  +289.026, Z    +0.000, E1   +70.567, E3 +43855.116}
SPL {X  -128.648, Y  +282.387, Z    +0.000, E1   +69.939, E3 +43862.931}
SPL {X  -125.063, Y  +277.720, Z    +0.000, E1   +69.378, E3 +43868.507}
SPL {X  -122.086, Y  +274.099, Z    +0.000, E1   +68.932, E3 +43872.752}
SPL {X   -84.117, Y  +241.407, Z    +0.000, E1   +58.224, E3 +43963.635}
ENDSPLINE

SPLINE
SPL {X  -106.708, Y  +258.294, Z    +0.000, E1   +53.789, E3 +44142.422}
SPL {X  -137.973, Y  +296.505, Z    +0.000, E1   +48.844, E3 +44181.202}
SPL {X  -154.359, Y  +335.426, Z    +0.000, E1   +34.338, E3 +44194.098}
SPL {X  -159.279, Y  +362.429, Z    +0.000, E1   +16.013, E3 +44197.698}
SPL {X  -159.976, Y  +375.387, Z    +0.000, E1    +4.229, E3 +44198.348}
SPL {X  -159.990, Y  +379.485, Z    +0.000, E1    +0.028, E3 +44198.394}
SPL {X  -159.990, Y  +381.270, Z    +0.000, E1    -3.383, E3 +44198.411}
SPL {X  -159.990, Y  +384.811, Z    +0.000, E1   -11.531, E3 +44198.501}
SPL {X  -159.990, Y  +390.180, Z    +0.000, E1   -24.142, E3 +44198.804}
SPL {X  -159.990, Y  +397.074, Z    +0.000, E1   -39.012, E3 +44199.414}
SPL {X  -159.990, Y  +405.152, Z    +0.000, E1   -50.697, E3 +44200.553}
SPL {X  -159.990, Y  +423.293, Z    +0.000, E1   -63.280, E3 +44204.554}
SPL {X  -159.990, Y  +493.649, Z    +0.000, E1   -71.671, E3 +44230.258}
SPL {X  -159.990, Y  +662.531, Z    +0.000, E1   -73.010, E3 +44317.081}
SPL {X  -159.805, Y  +684.185, Z    +0.000, E1   -72.979, E3 +44331.365}
SPL {X  -158.295, Y  +699.729, Z    +0.000, E1   -72.830, E3 +44343.036}
SPL {X  -155.857, Y  +712.630, Z    +0.000, E1   -72.572, E3 +44353.965}
SPL {X  -153.206, Y  +722.596, Z    +0.000, E1   -72.287, E3 +44363.146}
SPL {X  -150.445, Y  +730.933, Z    +0.000, E1   -71.979, E3 +44371.356}
SPL {X  -147.389, Y  +738.737, Z    +0.000, E1   -71.634, E3 +44379.429}
SPL {X  -144.044, Y  +746.129, Z    +0.000, E1   -71.236, E3 +44387.423}
SPL {X  -140.684, Y  +752.689, Z    +0.000, E1   -70.820, E3 +44394.798}
SPL {X  -137.335, Y  +758.572, Z    +0.000, E1   -70.388, E3 +44401.606}
SPL {X  -133.651, Y  +764.444, Z    +0.000, E1   -69.897, E3 +44408.558}
SPL {X  -129.492, Y  +770.461, Z    +0.000, E1   -69.311, E3 +44415.798}
SPL {X  -125.168, Y  +776.148, Z    +0.000, E1   -68.666, E3 +44422.674}
SPL {X  -122.036, Y  +779.960, Z    +0.000, E1   -68.144, E3 +44427.278}
SPL {X   -80.879, Y  +814.541, Z    +0.000, E1   -55.704, E3 +44548.595}
ENDSPLINE

SPLINE
SPL {X  -125.518, Y  +775.707, Z    +0.000, E1   -52.189, E3 +44720.073}
SPL {X  -150.797, Y  +729.951, Z    +0.000, E1   -39.777, E3 +44742.808}
SPL {X  -158.456, Y  +698.602, Z    +0.000, E1   -21.523, E3 +44748.510}
SPL {X  -159.738, Y  +685.469, Z    +0.000, E1   -10.595, E3 +44749.565}
SPL {X  -159.986, Y  +677.650, Z    +0.000, E1    -3.291, E3 +44749.819}
SPL {X  -159.990, Y  +674.500, Z    +0.000, E1    +0.000, E3 +44749.850}
SPL {X  -159.990, Y  +672.716, Z    +0.000, E1    +3.405, E3 +44749.866}
SPL {X  -159.990, Y  +668.521, Z    +0.000, E1   +13.007, E3 +44749.985}
SPL {X  -159.990, Y  +664.286, Z    +0.000, E1   +23.338, E3 +44750.217}
SPL {X  -159.990, Y  +658.431, Z    +0.000, E1   +35.998, E3 +44750.712}
SPL {X  -159.990, Y  +650.524, Z    +0.000, E1   +48.779, E3 +44751.700}
SPL {X  -159.990, Y  +641.022, Z    +0.000, E1   +57.726, E3 +44753.567}
SPL {X  -159.990, Y  +617.987, Z    +0.000, E1   +67.134, E3 +44759.463}
SPL {X  -159.990, Y  +532.407, Z    +0.000, E1   +73.084, E3 +44790.369}
SPL {X  -159.990, Y  +382.957, Z    +0.000, E1   +73.647, E3 +44866.629}
SPL {X  -159.615, Y  +366.548, Z    +0.000, E1   +73.602, E3 +44877.271}
SPL {X  -157.928, Y  +351.899, Z    +0.000, E1   +73.451, E3 +44888.126}
ENDSPLINE

SPLINE
SPL {X  -159.990, Y  +380.170, Z    +0.000, E1   +69.785, E3 +44904.266}
ENDSPLINE

SPLINE
SPL {X  -158.227, Y  +353.814, Z    +0.000, E1   +70.663, E3 +44916.159}
SPL {X  -154.257, Y  +335.055, Z    +0.000, E1   +71.089, E3 +44925.787}
SPL {X  -148.153, Y  +317.104, Z    +0.000, E1   +71.658, E3 +44932.933}
SPL {X  -143.479, Y  +306.716, Z    +0.000, E1   +71.847, E3 +44938.007}
SPL {X  -140.298, Y  +300.601, Z    +0.000, E1   +71.461, E3 +44944.762}
SPL {X  -137.001, Y  +294.872, Z    +0.000, E1   +71.048, E3 +44951.270}
SPL {X  -133.301, Y  +289.026, Z    +0.000, E1   +70.567, E3 +44958.057}
SPL {X  -128.648, Y  +282.387, Z    +0.000, E1   +69.939, E3 +44965.872}
SPL {X  -125.063, Y  +277.720, Z    +0.000, E1   +69.378, E3 +44971.448}
SPL {X  -122.086, Y  +274.099, Z    +0.000, E1   +68.932, E3 +44975.693}
SPL {X   -84.117, Y  +241.407, Z    +0.000, E1   +58.224, E3 +45066.576}
ENDSPLINE

SPLINE
SPL {X  -106.708, Y  +258.294, Z    +0.000, E1   +53.789, E3 +45245.363}
SPL {X  -137.973, Y  +296.505, Z    +0.000, E1   +48.844, E3 +45284.143}
SPL {X  -154.359, Y  +335.426, Z    +0.000, E1   +34.338, E3 +45297.039}
SPL {X  -159.279, Y  +362.429, Z    +0.000, E1   +16.013, E3 +45300.639}
SPL {X  -159.976, Y  +375.387, Z    +0.000, E1    +4.229, E3 +45301.290}
SPL {X  -159.990, Y  +379.485, Z    +0.000, E1    +0.028, E3 +45301.335}
SPL {X  -159.990, Y  +381.270, Z    +0.000, E1    -3.383, E3 +45301.352}
SPL {X  -159.990, Y  +384.811, Z    +0.000, E1   -11.531, E3 +45301.442}
SPL {X  -159.990, Y  +388.002, Z    +0.000, E1   -19.281, E3 +45301.592}
SPL {X  -159.990, Y  +394.075, Z    +0.000, E1   -32.836, E3 +45302.070}
SPL {X  -159.990, Y  +405.152, Z    +0.000, E1   -50.697, E3 +45303.494}
SPL {X  -159.990, Y  +423.293, Z    +0.000, E1   -63.280, E3 +45307.496}
SPL {X  -159.990, Y  +493.649, Z    +0.000, E1   -71.671, E3 +45333.199}
SPL {X  -159.990, Y  +662.531, Z    +0.000, E1   -73.010, E3 +45420.023}
SPL {X  -159.805, Y  +684.185, Z    +0.000, E1   -72.979, E3 +45434.307}
SPL {X  -158.739, Y  +696.464, Z    +0.000, E1   -72.862, E3 +45443.425}
SPL {X  -156.417, Y  +710.124, Z    +0.000, E1   -72.650, E3 +45454.649}
SPL {X  -153.206, Y  +722.596, Z    +0.000, E1   -72.287, E3 +45466.087}
SPL {X  -150.445, Y  +730.933, Z    +0.000, E1   -71.979, E3 +45474.297}
SPL {X  -147.389, Y  +738.737, Z    +0.000, E1   -71.634, E3 +45482.370}
SPL {X  -144.044, Y  +746.129, Z    +0.000, E1   -71.236, E3 +45490.364}
SPL {X  -140.684, Y  +752.689, Z    +0.000, E1   -70.820, E3 +45497.740}
SPL {X  -137.335, Y  +758.572, Z    +0.000, E1   -70.388, E3 +45504.547}
SPL {X  -134.566, Y  +763.037, Z    +0.000, E1   -70.007, E3 +45509.843}
SPL {X  -131.456, Y  +767.693, Z    +0.000, E1   -69.587, E3 +45515.407}
SPL {X  -127.440, Y  +773.226, Z    +0.000, E1   -69.006, E3 +45522.090}
SPL {X  -123.127, Y  +778.659, Z    +0.000, E1   -68.349, E3 +45528.632}
SPL {X   -80.879, Y  +814.541, Z    +0.000, E1   -55.704, E3 +45651.536}
ENDSPLINE

SPLINE
SPL {X  -125.518, Y  +775.707, Z    +0.000, E1   -52.189, E3 +45823.014}
SPL {X  -150.797, Y  +729.951, Z    +0.000, E1   -39.777, E3 +45845.749}
SPL {X  -158.456, Y  +698.602, Z    +0.000, E1   -21.523, E3 +45851.451}
SPL {X  -159.738, Y  +685.469, Z    +0.000, E1   -10.595, E3 +45852.506}
SPL {X  -159.986, Y  +677.650, Z    +0.000, E1    -3.291, E3 +45852.761}
SPL {X  -159.990, Y  +674.500, Z    +0.000, E1    +0.000, E3 +45852.791}
SPL {X  -159.990, Y  +672.716, Z    +0.000, E1    +3.405, E3 +45852.808}
SPL {X  -159.990, Y  +668.521, Z    +0.000, E1   +13.007, E3 +45852.927}
SPL {X  -159.990, Y  +662.839, Z    +0.000, E1   +26.519, E3 +45853.269}
SPL {X  -159.990, Y  +653.836, Z    +0.000, E1   +43.967, E3 +45854.199}
SPL {X  -159.990, Y  +641.022, Z    +0.000, E1   +57.726, E3 +45856.508}
SPL {X  -159.990, Y  +617.987, Z    +0.000, E1   +67.134, E3 +45862.404}
SPL {X  -159.990, Y  +532.407, Z    +0.000, E1   +73.084, E3 +45893.310}
SPL {X  -159.990, Y  +382.957, Z    +0.000, E1   +73.647, E3 +45969.570}
SPL {X  -159.196, Y  +361.585, Z    +0.000, E1   +73.581, E3 +45983.692}
SPL {X  -157.239, Y  +347.958, Z    +0.000, E1   +73.365, E3 +45994.287}
ENDSPLINE

SPLINE
SPL {X  -159.990, Y  +380.170, Z    +0.000, E1   +69.785, E3 +46007.207}
ENDSPLINE

SPLINE
SPL {X  -158.227, Y  +353.814, Z    +0.000, E1   +70.663, E3 +46019.101}
SPL {X  -155.560, Y  +340.111, Z    +0.000, E1   +70.976, E3 +46026.123}
SPL {X  -151.918, Y  +327.322, Z    +0.000, E1   +71.266, E3 +46032.466}
SPL {X  -144.697, Y  +309.238, Z    +0.000, E1   +71.848, E3 +46039.416}
SPL {X  -140.298, Y  +300.601, Z    +0.000, E1   +71.461, E3 +46047.703}
SPL {X  -137.001, Y  +294.872, Z    +0.000, E1   +71.048, E3 +46054.212}
SPL {X  -133.301, Y  +289.026, Z    +0.000, E1   +70.567, E3 +46060.998}
SPL {X  -129.603, Y  +283.692, Z    +0.000, E1   +70.051, E3 +46067.298}
SPL {X  -125.807, Y  +278.659, Z    +0.000, E1   +69.508, E3 +46073.257}
SPL {X  -122.086, Y  +274.099, Z    +0.000, E1   +68.932, E3 +46078.634}
SPL {X   -84.117, Y  +241.407, Z    +0.000, E1   +58.224, E3 +46169.517}
ENDSPLINE

SPLINE
SPL {X  -106.708, Y  +258.294, Z    +0.000, E1   +53.789, E3 +46348.304}
SPL {X  -137.973, Y  +296.505, Z    +0.000, E1   +48.844, E3 +46387.084}
SPL {X  -154.359, Y  +335.426, Z    +0.000, E1   +34.338, E3 +46399.980}
SPL {X  -159.279, Y  +362.429, Z    +0.000, E1   +16.013, E3 +46403.580}
SPL {X  -159.976, Y  +375.387, Z    +0.000, E1    +4.229, E3 +46404.231}
SPL {X  -159.990, Y  +379.485, Z    +0.000, E1    +0.028, E3 +46404.276}
SPL {X  -159.990, Y  +381.270, Z    +0.000, E1    -3.383, E3 +46404.293}
SPL {X  -159.990, Y  +386.246, Z    +0.000, E1   -14.704, E3 +46404.450}
SPL {X  -159.990, Y  +394.075, Z    +0.000, E1   -32.836, E3 +46405.011}
SPL {X  -159.990, Y  +405.152, Z    +0.000, E1   -50.697, E3 +46406.435}
SPL {X  -159.990, Y  +423.293, Z    +0.000, E1   -63.280, E3 +46410.437}
SPL {X  -159.990, Y  +493.649, Z    +0.000, E1   -71.671, E3 +46436.141}
SPL {X  -159.990, Y  +662.531, Z    +0.000, E1   -73.010, E3 +46522.964}
SPL {X  -159.805, Y  +684.185, Z    +0.000, E1   -72.979, E3 +46537.248}
SPL {X  -158.295, Y  +699.729, Z    +0.000, E1   -72.830, E3 +46548.918}
SPL {X  -155.857, Y  +712.630, Z    +0.000, E1   -72.572, E3 +46559.847}
SPL {X  -153.206, Y  +722.596, Z    +0.000, E1   -72.287, E3 +46569.028}
SPL {X  -150.445, Y  +730.933, Z    +0.000, E1   -71.979, E3 +46577.238}
SPL {X  -147.389, Y  +738.737, Z    +0.000, E1   -71.634, E3 +46585.311}
SPL {X  -144.044, Y  +746.129, Z    +0.000, E1   -71.236, E3 +46593.305}
SPL {X  -140.684, Y  +752.689, Z    +0.000, E1   -70.820, E3 +46600.681}
SPL {X  -136.099, Y  +760.606, Z    +0.000, E1   -70.253, E3 +46609.836}
SPL {X  -131.456, Y  +767.693, Z    +0.000, E1   -69.587, E3 +46618.348}
SPL {X  -127.440, Y  +773.226, Z    +0.000, E1   -69.006, E3 +46625.032}
SPL {X  -123.127, Y  +778.659, Z    +0.000, E1   -68.349, E3 +46631.574}
SPL {X   -80.879, Y  +814.541, Z    +0.000, E1   -55.704, E3 +46754.478}
ENDSPLINE

SPLINE
SPL {X  -125.518, Y  +775.707, Z    +0.000, E1   -52.189, E3 +46925.955}
SPL {X  -144.748, Y  +744.653, Z    +0.000, E1   -45.208, E3 +46944.151}
SPL {X  -153.147, Y  +722.791, Z    +0.000, E1   -36.417, E3 +46950.547}
SPL {X  -157.402, Y  +705.160, Z    +0.000, E1   -26.108, E3 +46953.642}
SPL {X  -159.480, Y  +689.270, Z    +0.000, E1   -14.023, E3 +46955.208}
SPL {X  -159.986, Y  +677.650, Z    +0.000, E1    -3.291, E3 +46955.702}
SPL {X  -159.990, Y  +674.500, Z    +0.000, E1    +0.000, E3 +46955.732}
SPL {X  -159.990, Y  +672.716, Z    +0.000, E1    +3.405, E3 +46955.749}
SPL {X  -159.990, Y  +668.521, Z    +0.000, E1   +13.007, E3 +46955.868}
SPL {X  -159.990, Y  +664.286, Z    +0.000, E1   +23.338, E3 +46956.099}
SPL {X  -159.990, Y  +658.431, Z    +0.000, E1   +35.998, E3 +46956.594}
SPL {X  -159.990, Y  +650.524, Z    +0.000, E1   +48.779, E3 +46957.582}
SPL {X  -159.990, Y  +641.022, Z    +0.000, E1   +57.726, E3 +46959.449}
SPL {X  -159.990, Y  +617.987, Z    +0.000, E1   +67.134, E3 +46965.345}
SPL {X  -159.990, Y  +532.407, Z    +0.000, E1   +73.084, E3 +46996.252}
SPL {X  -159.990, Y  +390.607, Z    +0.000, E1   +73.632, E3 +47067.788}
SPL {X  -159.886, Y  +371.742, Z    +0.000, E1   +73.650, E3 +47079.574}
SPL {X  -157.928, Y  +351.899, Z    +0.000, E1   +73.451, E3 +47094.008}
ENDSPLINE

SPLINE
SPL {X  -159.990, Y  +380.170, Z    +0.000, E1   +69.785, E3 +47110.148}
ENDSPLINE

SPLINE
SPL {X  -158.227, Y  +353.814, Z    +0.000, E1   +70.663, E3 +47122.042}
SPL {X  -155.560, Y  +340.111, Z    +0.000, E1   +70.976, E3 +47129.064}
SPL {X  -151.918, Y  +327.322, Z    +0.000, E1   +71.266, E3 +47135.407}
SPL {X  -144.697, Y  +309.238, Z    +0.000, E1   +71.848, E3 +47142.357}
SPL {X  -140.298, Y  +300.601, Z    +0.000, E1   +71.461, E3 +47150.644}
SPL {X  -135.903, Y  +293.078, Z    +0.000, E1   +70.930, E3 +47159.182}
SPL {X  -132.382, Y  +287.656, Z    +0.000, E1   +70.425, E3 +47165.574}
SPL {X  -128.648, Y  +282.387, Z    +0.000, E1   +69.939, E3 +47171.755}
SPL {X  -125.063, Y  +277.720, Z    +0.000, E1   +69.378, E3 +47177.330}
SPL {X  -122.086, Y  +274.099, Z    +0.000, E1   +68.932, E3 +47181.576}
SPL {X   -84.117, Y  +241.407, Z    +0.000, E1   +58.224, E3 +47272.458}
ENDSPLINE

SPLINE
SPL {X  -106.708, Y  +258.294, Z    +0.000, E1   +53.789, E3 +47451.245}
SPL {X  -137.973, Y  +296.505, Z    +0.000, E1   +48.844, E3 +47490.025}
SPL {X  -154.359, Y  +335.426, Z    +0.000, E1   +34.338, E3 +47502.921}
SPL {X  -159.279, Y  +362.429, Z    +0.000, E1   +16.013, E3 +47506.521}
SPL {X  -159.976, Y  +375.387, Z    +0.000, E1    +4.229, E3 +47507.172}
SPL {X  -159.990, Y  +379.485, Z    +0.000, E1    +0.028, E3 +47507.217}
SPL {X  -159.990, Y  +381.270, Z    +0.000, E1    -3.383, E3 +47507.234}
SPL {X  -159.990, Y  +384.811, Z    +0.000, E1   -11.531, E3 +47507.324}
SPL {X  -159.990, Y  +390.180, Z    +0.000, E1   -24.142, E3 +47507.627}
SPL {X  -159.990, Y  +397.074, Z    +0.000, E1   -39.012, E3 +47508.237}
SPL {X  -159.990, Y  +405.152, Z    +0.000, E1   -50.697, E3 +47509.377}
SPL {X  -159.990, Y  +423.293, Z    +0.000, E1   -63.280, E3 +47513.378}
SPL {X  -159.990, Y  +493.649, Z    +0.000, E1   -71.671, E3 +47539.082}
SPL {X  -159.990, Y  +662.531, Z    +0.000, E1   -73.010, E3 +47625.905}
SPL {X  -159.805, Y  +684.185, Z    +0.000, E1   -72.979, E3 +47640.189}
SPL {X  -158.739, Y  +696.464, Z    +0.000, E1   -72.862, E3 +47649.308}
SPL {X  -156.417, Y  +710.124, Z    +0.000, E1   -72.650, E3 +47660.531}
SPL {X  -153.206, Y  +722.596, Z    +0.000, E1   -72.287, E3 +47671.969}
SPL {X  -150.445, Y  +730.933, Z    +0.000, E1   -71.979, E3 +47680.179}
SPL {X  -147.389, Y  +738.737, Z    +0.000, E1   -71.634, E3 +47688.252}
SPL {X  -144.044, Y  +746.129, Z    +0.000, E1   -71.236, E3 +47696.247}
SPL {X  -140.684, Y  +752.689, Z    +0.000, E1   -70.820, E3 +47703.622}
SPL {X  -137.335, Y  +758.572, Z    +0.000, E1   -70.388, E3 +47710.429}
SPL {X  -134.566, Y  +763.037, Z    +0.000, E1   -70.007, E3 +47715.725}
SPL {X  -131.456, Y  +767.693, Z    +0.000, E1   -69.587, E3 +47721.289}
SPL {X  -127.440, Y  +773.226, Z    +0.000, E1   -69.006, E3 +47727.973}
SPL {X  -123.127, Y  +778.659, Z    +0.000, E1   -68.349, E3 +47734.515}
SPL {X   -80.879, Y  +814.541, Z    +0.000, E1   -55.704, E3 +47857.419}
ENDSPLINE

SPLINE
SPL {X  -125.518, Y  +775.707, Z    +0.000, E1   -52.189, E3 +48028.896}
SPL {X  -144.748, Y  +744.653, Z    +0.000, E1   -45.208, E3 +48047.092}
SPL {X  -153.147, Y  +722.791, Z    +0.000, E1   -36.417, E3 +48053.488}
SPL {X  -157.402, Y  +705.160, Z    +0.000, E1   -26.108, E3 +48056.583}
SPL {X  -159.480, Y  +689.270, Z    +0.000, E1   -14.023, E3 +48058.149}
SPL {X  -159.986, Y  +677.650, Z    +0.000, E1    -3.291, E3 +48058.643}
SPL {X  -159.990, Y  +674.500, Z    +0.000, E1    +0.000, E3 +48058.673}
SPL {X  -159.990, Y  +672.716, Z    +0.000, E1    +3.405, E3 +48058.690}
SPL {X  -159.990, Y  +668.521, Z    +0.000, E1   +13.007, E3 +48058.809}
SPL {X  -159.990, Y  +662.839, Z    +0.000, E1   +26.519, E3 +48059.151}
SPL {X  -159.990, Y  +653.836, Z    +0.000, E1   +43.967, E3 +48060.082}
SPL {X  -159.990, Y  +641.022, Z    +0.000, E1   +57.726, E3 +48062.391}
SPL {X  -159.990, Y  +617.987, Z    +0.000, E1   +67.134, E3 +48068.286}
SPL {X  -159.990, Y  +532.407, Z    +0.000, E1   +73.084, E3 +48099.193}
SPL {X  -159.990, Y  +382.957, Z    +0.000, E1   +73.647, E3 +48175.452}
SPL {X  -159.615, Y  +366.548, Z    +0.000, E1   +73.602, E3 +48186.095}
SPL {X  -157.928, Y  +351.899, Z    +0.000, E1   +73.451, E3 +48196.949}
ENDSPLINE

SPLINE
SPL {X  -159.990, Y  +380.170, Z    +0.000, E1   +69.785, E3 +48213.089}
ENDSPLINE

SPLINE
SPL {X  -158.227, Y  +353.814, Z    +0.000, E1   +70.663, E3 +48224.983}
SPL {X  -155.560, Y  +340.111, Z    +0.000, E1   +70.976, E3 +48232.005}
SPL {X  -151.918, Y  +327.322, Z    +0.000, E1   +71.266, E3 +48238.349}
SPL {X  -144.697, Y  +309.238, Z    +0.000, E1   +71.848, E3 +48245.298}
SPL {X  -140.298, Y  +300.601, Z    +0.000, E1   +71.461, E3 +48253.586}
SPL {X  -135.903, Y  +293.078, Z    +0.000, E1   +70.930, E3 +48262.123}
SPL {X  -130.487, Y  +284.926, Z    +0.000, E1   +70.202, E3 +48271.683}
SPL {X  -125.807, Y  +278.659, Z    +0.000, E1   +69.508, E3 +48279.139}
SPL {X  -122.967, Y  +275.148, Z    +0.000, E1   +69.053, E3 +48283.308}
SPL {X  -121.236, Y  +273.103, Z    +0.000, E1   +68.779, E3 +48285.694}
SPL {X   -84.117, Y  +241.407, Z    +0.000, E1   +58.224, E3 +48375.399}
ENDSPLINE

SPLINE
SPL {X  -106.708, Y  +258.294, Z    +0.000, E1   +53.789, E3 +48554.186}
SPL {X  -137.973, Y  +296.505, Z    +0.000, E1   +48.844, E3 +48592.966}
SPL {X  -154.359, Y  +335.426, Z    +0.000, E1   +34.338, E3 +48605.862}
SPL {X  -159.279, Y  +362.429, Z    +0.000, E1   +16.013, E3 +48609.462}
SPL {X  -159.976, Y  +375.387, Z    +0.000, E1    +4.229, E3 +48610.113}
SPL {X  -159.990, Y  +379.485, Z    +0.000, E1    +0.028, E3 +48610.158}
SPL {X  -159.990, Y  +381.270, Z    +0.000, E1    -3.383, E3 +48610.175}
SPL {X  -159.990, Y  +386.246, Z    +0.000, E1   -14.704, E3 +48610.333}
SPL {X  -159.990, Y  +394.075, Z    +0.000, E1   -32.836, E3 +48610.894}
SPL {X  -159.990, Y  +405.152, Z    +0.000, E1   -50.697, E3 +48612.318}
SPL {X  -159.990, Y  +423.293, Z    +0.000, E1   -63.280, E3 +48616.319}
SPL {X  -159.990, Y  +493.649, Z    +0.000, E1   -71.671, E3 +48642.023}
SPL {X  -159.990, Y  +662.531, Z    +0.000, E1   -73.010, E3 +48728.846}
SPL {X  -159.805, Y  +684.185, Z    +0.000, E1   -72.979, E3 +48743.130}
SPL {X  -158.295, Y  +699.729, Z    +0.000, E1   -72.830, E3 +48754.800}
SPL {X  -155.857, Y  +712.630, Z    +0.000, E1   -72.572, E3 +48765.729}
SPL {X  -153.206, Y  +722.596, Z    +0.000, E1   -72.287, E3 +48774.910}
SPL {X  -150.445, Y  +730.933, Z    +0.000, E1   -71.979, E3 +48783.121}
SPL {X  -147.389, Y  +738.737, Z    +0.000, E1   -71.634, E3 +48791.193}
SPL {X  -144.044, Y  +746.129, Z    +0.000, E1   -71.236, E3 +48799.188}
SPL {X  -140.684, Y  +752.689, Z    +0.000, E1   -70.820, E3 +48806.563}
SPL {X  -137.335, Y  +758.572, Z    +0.000, E1   -70.388, E3 +48813.370}
SPL {X  -133.651, Y  +764.444, Z    +0.000, E1   -69.897, E3 +48820.322}
SPL {X  -129.492, Y  +770.461, Z    +0.000, E1   -69.311, E3 +48827.563}
SPL {X  -125.168, Y  +776.148, Z    +0.000, E1   -68.666, E3 +48834.439}
SPL {X  -122.036, Y  +779.960, Z    +0.000, E1   -68.144, E3 +48839.042}
SPL {X   -80.879, Y  +814.541, Z    +0.000, E1   -55.704, E3 +48960.360}
ENDSPLINE

SPLINE
SPL {X  -125.518, Y  +775.707, Z    +0.000, E1   -52.189, E3 +49131.837}
SPL {X  -144.748, Y  +744.653, Z    +0.000, E1   -45.208, E3 +49150.033}
SPL {X  -153.147, Y  +722.791, Z    +0.000, E1   -36.417, E3 +49156.429}
SPL {X  -157.402, Y  +705.160, Z    +0.000, E1   -26.108, E3 +49159.524}
SPL {X  -159.480, Y  +689.270, Z    +0.000, E1   -14.023, E3 +49161.090}
SPL {X  -159.986, Y  +677.650, Z    +0.000, E1    -3.291, E3 +49161.584}
SPL {X  -159.990, Y  +674.500, Z    +0.000, E1    +0.000, E3 +49161.615}
SPL {X  -159.990, Y  +672.716, Z    +0.000, E1    +3.405, E3 +49161.631}
SPL {X  -159.990, Y  +668.521, Z    +0.000, E1   +13.007, E3 +49161.750}
SPL {X  -159.990, Y  +664.286, Z    +0.000, E1   +23.338, E3 +49161.982}
SPL {X  -159.990, Y  +658.431, Z    +0.000, E1   +35.998, E3 +49162.476}
SPL {X  -159.990, Y  +650.524, Z    +0.000, E1   +48.779, E3 +49163.465}
SPL {X  -159.990, Y  +641.022, Z    +0.000, E1   +57.726, E3 +49165.332}
SPL {X  -159.990, Y  +617.987, Z    +0.000, E1   +67.134, E3 +49171.227}
SPL {X  -159.990, Y  +532.407, Z    +0.000, E1   +73.084, E3 +49202.134}
SPL {X  -159.990, Y  +390.607, Z    +0.000, E1   +73.632, E3 +49273.670}
SPL {X  -159.886, Y  +371.742, Z    +0.000, E1   +73.650, E3 +49285.457}
SPL {X  -157.928, Y  +351.899, Z    +0.000, E1   +73.451, E3 +49299.890}
ENDSPLINE

SPLINE
SPL {X  -159.990, Y  +380.170, Z    +0.000, E1   +69.785, E3 +49316.031}
ENDSPLINE

SPLINE
SPL {X  -158.227, Y  +353.814, Z    +0.000, E1   +70.663, E3 +49327.924}
SPL {X  -155.560, Y  +340.111, Z    +0.000, E1   +70.976, E3 +49334.946}
SPL {X  -151.918, Y  +327.322, Z    +0.000, E1   +71.266, E3 +49341.290}
SPL {X  -144.697, Y  +309.238, Z    +0.000, E1   +71.848, E3 +49348.239}
SPL {X  -140.298, Y  +300.601, Z    +0.000, E1   +71.461, E3 +49356.527}
SPL {X  -137.001, Y  +294.872, Z    +0.000, E1   +71.048, E3 +49363.035}
SPL {X  -133.301, Y  +289.026, Z    +0.000, E1   +70.567, E3 +49369.822}
SPL {X  -129.603, Y  +283.692, Z    +0.000, E1   +70.051, E3 +49376.122}
SPL {X  -125.807, Y  +278.659, Z    +0.000, E1   +69.508, E3 +49382.080}
SPL {X  -122.086, Y  +274.099, Z    +0.000, E1   +68.932, E3 +49387.458}
SPL {X   -84.117, Y  +241.407, Z    +0.000, E1   +58.224, E3 +49478.341}
ENDSPLINE

SPLINE
SPL {X  -106.708, Y  +258.294, Z    +0.000, E1   +53.789, E3 +49657.127}
SPL {X  -137.973, Y  +296.505, Z    +0.000, E1   +48.844, E3 +49695.908}
SPL {X  -154.359, Y  +335.426, Z    +0.000, E1   +34.338, E3 +49708.804}
SPL {X  -159.279, Y  +362.429, Z    +0.000, E1   +16.013, E3 +49712.404}
SPL {X  -159.976, Y  +375.387, Z    +0.000, E1    +4.229, E3 +49713.054}
SPL {X  -159.990, Y  +379.485, Z    +0.000, E1    +0.028, E3 +49713.099}
SPL {X  -159.990, Y  +381.270, Z    +0.000, E1    -3.383, E3 +49713.117}
SPL {X  -159.990, Y  +386.246, Z    +0.000, E1   -14.704, E3 +49713.274}
SPL {X  -159.990, Y  +394.075, Z    +0.000, E1   -32.836, E3 +49713.835}
SPL {X  -159.990, Y  +405.152, Z    +0.000, E1   -50.697, E3 +49715.259}
SPL {X  -159.990, Y  +423.293, Z    +0.000, E1   -63.280, E3 +49719.260}
SPL {X  -159.990, Y  +493.649, Z    +0.000, E1   -71.671, E3 +49744.964}
SPL {X  -159.990, Y  +662.531, Z    +0.000, E1   -73.010, E3 +49831.787}
SPL {X  -159.805, Y  +684.185, Z    +0.000, E1   -72.979, E3 +49846.071}
SPL {X  -158.295, Y  +699.729, Z    +0.000, E1   -72.830, E3 +49857.742}
SPL {X  -155.857, Y  +712.630, Z    +0.000, E1   -72.572, E3 +49868.671}
SPL {X  -153.206, Y  +722.596, Z    +0.000, E1   -72.287, E3 +49877.851}
SPL {X  -150.445, Y  +730.933, Z    +0.000, E1   -71.979, E3 +49886.062}
SPL {X  -147.389, Y  +738.737, Z    +0.000, E1   -71.634, E3 +49894.135}
SPL {X  -144.044, Y  +746.129, Z    +0.000, E1   -71.236, E3 +49902.129}
SPL {X  -140.684, Y  +752.689, Z    +0.000, E1   -70.820, E3 +49909.504}
SPL {X  -136.099, Y  +760.606, Z    +0.000, E1   -70.253, E3 +49918.660}
SPL {X  -131.456, Y  +767.693, Z    +0.000, E1   -69.587, E3 +49927.171}
SPL {X  -127.440, Y  +773.226, Z    +0.000, E1   -69.006, E3 +49933.855}
SPL {X  -123.127, Y  +778.659, Z    +0.000, E1   -68.349, E3 +49940.397}
SPL {X   -80.879, Y  +814.541, Z    +0.000, E1   -55.704, E3 +50063.301}
ENDSPLINE

SPLINE
SPL {X  -125.518, Y  +775.707, Z    +0.000, E1   -52.189, E3 +50234.779}
SPL {X  -150.797, Y  +729.951, Z    +0.000, E1   -39.777, E3 +50257.514}
SPL {X  -157.402, Y  +705.160, Z    +0.000, E1   -26.108, E3 +50262.465}
SPL {X  -159.480, Y  +689.270, Z    +0.000, E1   -14.023, E3 +50264.031}
SPL {X  -159.986, Y  +677.650, Z    +0.000, E1    -3.291, E3 +50264.525}
SPL {X  -159.990, Y  +674.500, Z    +0.000, E1    +0.000, E3 +50264.556}
SPL {X  -159.990, Y  +672.716, Z    +0.000, E1    +3.405, E3 +50264.572}
SPL {X  -159.990, Y  +668.521, Z    +0.000, E1   +13.007, E3 +50264.691}
SPL {X  -159.990, Y  +662.839, Z    +0.000, E1   +26.519, E3 +50265.034}
SPL {X  -159.990, Y  +653.836, Z    +0.000, E1   +43.967, E3 +50265.964}
SPL {X  -159.990, Y  +641.022, Z    +0.000, E1   +57.726, E3 +50268.273}
SPL {X  -159.990, Y  +617.987, Z    +0.000, E1   +67.134, E3 +50274.168}
SPL {X  -159.990, Y  +532.407, Z    +0.000, E1   +73.084, E3 +50305.075}
SPL {X  -159.990, Y  +390.607, Z    +0.000, E1   +73.632, E3 +50376.611}
SPL {X  -159.886, Y  +371.742, Z    +0.000, E1   +73.650, E3 +50388.398}
SPL {X  -157.928, Y  +351.899, Z    +0.000, E1   +73.451, E3 +50402.832}
ENDSPLINE

SPLINE
SPL {X  -159.990, Y  +380.170, Z    +0.000, E1   +69.785, E3 +50418.972}
ENDSPLINE

SPLINE
SPL {X  -158.227, Y  +353.814, Z    +0.000, E1   +70.663, E3 +50430.865}
SPL {X  -155.560, Y  +340.111, Z    +0.000, E1   +70.976, E3 +50437.887}
SPL {X  -151.918, Y  +327.322, Z    +0.000, E1   +71.266, E3 +50444.231}
SPL {X  -144.697, Y  +309.238, Z    +0.000, E1   +71.848, E3 +50451.181}
SPL {X  -140.298, Y  +300.601, Z    +0.000, E1   +71.461, E3 +50459.468}
SPL {X  -135.903, Y  +293.078, Z    +0.000, E1   +70.930, E3 +50468.006}
SPL {X  -130.487, Y  +284.926, Z    +0.000, E1   +70.202, E3 +50477.565}
SPL {X  -125.807, Y  +278.659, Z    +0.000, E1   +69.508, E3 +50485.022}
SPL {X  -122.967, Y  +275.148, Z    +0.000, E1   +69.053, E3 +50489.190}
SPL {X  -121.236, Y  +273.103, Z    +0.000, E1   +68.779, E3 +50491.576}
SPL {X   -84.117, Y  +241.407, Z    +0.000, E1   +58.224, E3 +50581.282}
ENDSPLINE

SPLINE
SPL {X  -116.986, Y  +268.362, Z    +0.000, E1   +53.233, E3 +50775.197}
SPL {X  -146.319, Y  +312.789, Z    +0.000, E1   +44.152, E3 +50805.663}
SPL {X  -157.053, Y  +346.986, Z    +0.000, E1   +27.437, E3 +50813.695}
SPL {X  -159.518, Y  +365.226, Z    +0.000, E1   +13.562, E3 +50815.560}
SPL {X  -159.976, Y  +375.387, Z    +0.000, E1    +4.229, E3 +50815.996}
SPL {X  -159.990, Y  +379.485, Z    +0.000, E1    +0.028, E3 +50816.041}
SPL {X  -159.990, Y  +381.270, Z    +0.000, E1    -3.383, E3 +50816.058}
SPL {X  -159.990, Y  +386.246, Z    +0.000, E1   -14.704, E3 +50816.215}
SPL {X  -159.990, Y  +394.075, Z    +0.000, E1   -32.836, E3 +50816.776}
SPL {X  -159.990, Y  +405.152, Z    +0.000, E1   -50.697, E3 +50818.200}
SPL {X  -159.990, Y  +423.293, Z    +0.000, E1   -63.280, E3 +50822.201}
SPL {X  -159.990, Y  +493.649, Z    +0.000, E1   -71.671, E3 +50847.905}
SPL {X  -159.990, Y  +662.531, Z    +0.000, E1   -73.010, E3 +50934.728}
SPL {X  -159.805, Y  +684.185, Z    +0.000, E1   -72.979, E3 +50949.012}
SPL {X  -158.295, Y  +699.729, Z    +0.000, E1   -72.830, E3 +50960.683}
SPL {X  -155.857, Y  +712.630, Z    +0.000, E1   -72.572, E3 +50971.612}
SPL {X  -153.206, Y  +722.596, Z    +0.000, E1   -72.287, E3 +50980.793}
SPL {X  -150.445, Y  +730.933, Z    +0.000, E1   -71.979, E3 +50989.003}
SPL {X  -147.389, Y  +738.737, Z    +0.000, E1   -71.634, E3 +50997.076}
SPL {X  -144.044, Y  +746.129, Z    +0.000, E1   -71.236, E3 +51005.070}
SPL {X  -140.684, Y  +752.689, Z    +0.000, E1   -70.820, E3 +51012.445}
SPL {X  -136.099, Y  +760.606, Z    +0.000, E1   -70.253, E3 +51021.601}
SPL {X  -131.456, Y  +767.693, Z    +0.000, E1   -69.587, E3 +51030.113}
SPL {X  -127.440, Y  +773.226, Z    +0.000, E1   -69.006, E3 +51036.796}
SPL {X  -123.127, Y  +778.659, Z    +0.000, E1   -68.349, E3 +51043.338}
SPL {X   -80.879, Y  +814.541, Z    +0.000, E1   -55.704, E3 +51166.242}
ENDSPLINE

SPLINE
SPL {X  -125.518, Y  +775.707, Z    +0.000, E1   -52.189, E3 +51337.720}
SPL {X  -150.797, Y  +729.951, Z    +0.000, E1   -39.777, E3 +51360.455}
SPL {X  -158.456, Y  +698.602, Z    +0.000, E1   -21.523, E3 +51366.157}
SPL {X  -159.738, Y  +685.469, Z    +0.000, E1   -10.595, E3 +51367.212}
SPL {X  -159.986, Y  +677.650, Z    +0.000, E1    -3.291, E3 +51367.467}
SPL {X  -159.990, Y  +674.500, Z    +0.000, E1    +0.000, E3 +51367.497}
SPL {X  -159.990, Y  +672.716, Z    +0.000, E1    +3.405, E3 +51367.513}
SPL {X  -159.990, Y  +668.521, Z    +0.000, E1   +13.007, E3 +51367.633}
SPL {X  -159.990, Y  +662.839, Z    +0.000, E1   +26.519, E3 +51367.975}
SPL {X  -159.990, Y  +653.836, Z    +0.000, E1   +43.967, E3 +51368.905}
SPL {X  -159.990, Y  +641.022, Z    +0.000, E1   +57.726, E3 +51371.214}
SPL {X  -159.990, Y  +617.987, Z    +0.000, E1   +67.134, E3 +51377.110}
SPL {X  -159.990, Y  +532.407, Z    +0.000, E1   +73.084, E3 +51408.016}
SPL {X  -159.990, Y  +382.957, Z    +0.000, E1   +73.647, E3 +51484.276}
SPL {X  -159.615, Y  +366.548, Z    +0.000, E1   +73.602, E3 +51494.918}
SPL {X  -157.928, Y  +351.899, Z    +0.000, E1   +73.451, E3 +51505.773}
ENDSPLINE

SPLINE
SPL {X  -159.990, Y  +380.170, Z    +0.000, E1   +69.785, E3 +51521.913}
ENDSPLINE

